C01819=1039.319,-74.831,422.675,168.772,36.713,156.907
C01820=1039.313,-75.080,422.686,168.769,36.713,156.907
C01821=1039.306,-75.330,422.697,168.767,36.713,156.907
C01822=1039.301,-75.580,422.708,168.764,36.713,156.907
C01823=1039.294,-75.829,422.720,168.762,36.713,156.907
C01824=1039.288,-76.079,422.731,168.759,36.713,156.907
C01825=1039.282,-76.329,422.742,168.757,36.713,156.907
C01826=1039.276,-76.578,422.754,168.754,36.713,156.907
C01827=1039.269,-76.828,422.765,168.752,36.714,156.907
C01828=1039.264,-77.077,422.776,168.749,36.714,156.907
C01829=1039.257,-77.328,422.787,168.747,36.714,156.907
C01830=1039.251,-77.576,422.799,168.745,36.714,156.907
C01831=1039.244,-77.826,422.810,168.742,36.714,156.907
C01832=1039.238,-78.076,422.820,168.740,36.714,156.907
C01833=1039.232,-78.326,422.832,168.737,36.714,156.907
C01834=1039.226,-78.575,422.843,168.735,36.714,156.907
C01835=1039.220,-78.825,422.854,168.732,36.714,156.907
C01836=1039.214,-79.075,422.865,168.730,36.714,156.907
C01837=1039.208,-79.325,422.877,168.727,36.714,156.907
C01838=1039.202,-79.574,422.887,168.725,36.714,156.907
C01839=1039.196,-79.824,422.899,168.722,36.714,156.907
C01840=1039.190,-80.074,422.910,168.720,36.714,156.907
C01841=1039.182,-80.323,422.921,168.717,36.714,156.907
C01842=1039.177,-80.573,422.932,168.715,36.714,156.907
C01843=1039.170,-80.823,422.943,168.712,36.714,156.907
C01844=1039.164,-81.072,422.953,168.710,36.714,156.907
C01845=1039.158,-81.321,422.964,168.707,36.715,156.907
C01846=1039.152,-81.572,422.975,168.705,36.715,156.907
C01847=1039.145,-81.821,422.986,168.702,36.715,156.907
C01848=1039.139,-82.071,422.997,168.700,36.715,156.907
C01849=1039.133,-82.321,423.008,168.697,36.716,156.908
C01850=1039.126,-82.570,423.019,168.695,36.716,156.908
C01851=1039.120,-82.820,423.029,168.692,36.716,156.908
C01852=1039.114,-83.070,423.041,168.690,36.716,156.908
C01853=1039.108,-83.319,423.051,168.687,36.716,156.908
C01854=1039.101,-83.605,423.064,168.684,36.716,156.908
C01855=1039.094,-83.889,423.076,168.682,36.717,156.908
C01856=1039.087,-84.174,423.089,168.679,36.717,156.908
C01857=1039.080,-84.459,423.101,168.676,36.717,156.908
C01858=1039.073,-84.709,423.111,168.673,36.717,156.908
C01859=1039.067,-84.958,423.122,168.672,36.718,156.908
C01860=1039.061,-85.209,423.133,168.669,36.718,156.908
C01861=1039.054,-85.458,423.144,168.667,36.718,156.908
C01862=1039.049,-85.707,423.155,168.664,36.718,156.908
C01863=1039.042,-85.957,423.166,168.662,36.719,156.908
C01864=1039.036,-86.207,423.175,168.659,36.719,156.908
C01865=1039.030,-86.457,423.186,168.657,36.719,156.908
C01866=1039.024,-86.707,423.198,168.654,36.719,156.908
C01867=1039.018,-86.956,423.208,168.652,36.719,156.908
C01868=1039.012,-87.206,423.219,168.649,36.719,156.908
C01869=1039.005,-87.456,423.230,168.647,36.719,156.908
C01870=1038.999,-87.705,423.240,168.644,36.720,156.908
C01871=1038.993,-87.954,423.251,168.642,36.720,156.908
C01872=1038.986,-88.205,423.261,168.639,36.720,156.908
C01873=1038.981,-88.454,423.272,168.637,36.721,156.908
C01874=1038.975,-88.704,423.283,168.634,36.721,156.908
C01875=1038.968,-88.954,423.293,168.631,36.721,156.908
C01876=1038.962,-89.203,423.304,168.629,36.721,156.908
C01877=1038.957,-89.453,423.315,168.626,36.721,156.908
C01878=1038.950,-89.703,423.325,168.624,36.721,156.908
C01879=1038.944,-89.953,423.336,168.621,36.722,156.908
C01880=1038.937,-90.202,423.346,168.619,36.722,156.908
C01881=1038.932,-90.451,423.357,168.616,36.722,156.908
C01882=1038.926,-90.702,423.368,168.614,36.723,156.909
C01883=1038.919,-90.951,423.378,168.611,36.723,156.909
C01884=1038.913,-91.201,423.389,168.609,36.723,156.909
C01885=1038.907,-91.450,423.399,168.606,36.723,156.909
C01886=1038.902,-91.700,423.409,168.604,36.723,156.909
C01887=1038.895,-91.950,423.421,168.601,36.724,156.909
C01888=1038.889,-92.200,423.431,168.599,36.724,156.909
C01889=1038.883,-92.450,423.441,168.596,36.724,156.909
C01890=1038.877,-92.699,423.451,168.593,36.725,156.909
C01891=1038.870,-92.949,423.463,168.591,36.725,156.909
C01892=1038.864,-93.199,423.472,168.588,36.725,156.909
C01893=1038.859,-93.448,423.483,168.586,36.726,156.909
C01894=1038.853,-93.698,423.494,168.583,36.726,156.909
C01895=1038.847,-93.948,423.503,168.581,36.726,156.909
C01896=1038.841,-94.197,423.514,168.578,36.726,156.909
C01897=1038.834,-94.447,423.525,168.576,36.726,156.909
C01898=1038.828,-94.697,423.535,168.573,36.727,156.909
C01899=1038.823,-94.947,423.546,168.571,36.727,156.909
C01900=1038.816,-95.196,423.556,168.568,36.727,156.909
C01901=1038.811,-95.446,423.566,168.566,36.728,156.909
C01902=1038.804,-95.695,423.577,168.563,36.728,156.909
C01903=1038.799,-95.945,423.587,168.561,36.728,156.909
C01904=1038.792,-96.195,423.598,168.559,36.728,156.909
C01905=1038.786,-96.445,423.608,168.556,36.728,156.909
C01906=1038.780,-96.694,423.618,168.554,36.729,156.909
C01907=1038.774,-96.944,423.628,168.551,36.729,156.909
C01908=1038.769,-97.194,423.639,168.549,36.730,156.910
C01909=1038.762,-97.443,423.649,168.546,36.730,156.910
C01910=1038.756,-97.693,423.659,168.544,36.730,156.910
C01911=1038.751,-97.943,423.669,168.541,36.730,156.910
C01912=1038.744,-98.193,423.680,168.538,36.731,156.910
C01913=1038.737,-98.443,423.689,168.536,36.731,156.910
C01914=1038.732,-98.692,423.700,168.533,36.732,156.910
C01915=1038.725,-98.942,423.710,168.531,36.732,156.910
C01916=1038.719,-99.191,423.720,168.528,36.732,156.910
C01917=1038.714,-99.441,423.730,168.525,36.733,156.910
C01918=1038.706,-99.729,423.741,168.522,36.734,156.910
C01919=1038.699,-100.015,423.753,168.519,36.734,156.910
C01920=1038.692,-100.303,423.765,168.517,36.734,156.910
C01921=1038.685,-100.590,423.776,168.514,36.735,156.910
C01922=1038.679,-100.840,423.786,168.511,36.735,156.910
C01923=1038.673,-101.089,423.797,168.508,36.736,156.911
C01924=1038.667,-101.339,423.806,168.506,36.737,156.911
C01925=1038.660,-101.589,423.816,168.503,36.737,156.911
C01926=1038.655,-101.839,423.827,168.501,36.737,156.911
C01927=1038.649,-102.088,423.836,168.498,36.737,156.911
C01928=1038.642,-102.338,423.846,168.495,36.738,156.911
C01929=1038.636,-102.587,423.856,168.494,36.739,156.911
C01930=1038.630,-102.837,423.866,168.491,36.739,156.911
C01931=1038.624,-103.087,423.876,168.489,36.739,156.911
C01932=1038.618,-103.336,423.886,168.486,36.740,156.911
C01933=1038.612,-103.587,423.896,168.483,36.740,156.911
C01934=1038.606,-103.836,423.906,168.481,36.741,156.911
C01935=1038.600,-104.086,423.916,168.478,36.741,156.911
C01936=1038.594,-104.335,423.926,168.476,36.741,156.911
C01937=1038.588,-104.585,423.936,168.473,36.742,156.911
C01938=1038.582,-104.835,423.946,168.470,36.743,156.912
C01939=1038.576,-105.085,423.955,168.468,36.743,156.912
C01940=1038.570,-105.335,423.965,168.465,36.743,156.912
C01941=1038.564,-105.584,423.976,168.463,36.744,156.912
C01942=1038.558,-105.834,423.985,168.460,36.745,156.912
C01943=1038.552,-106.084,423.995,168.457,36.745,156.912
C01944=1038.545,-106.334,424.004,168.455,36.745,156.912
C01945=1038.539,-106.583,424.014,168.452,36.746,156.912
C01946=1038.533,-106.833,424.025,168.449,36.747,156.912
C01947=1038.527,-107.083,424.034,168.447,36.747,156.912
C01948=1038.521,-107.333,424.044,168.444,36.747,156.912
C01949=1038.515,-107.582,424.053,168.442,36.748,156.912
C01950=1038.509,-107.832,424.063,168.440,36.749,156.913
C01951=1038.503,-108.082,424.073,168.437,36.749,156.913
C01952=1038.496,-108.332,424.082,168.435,36.749,156.913
C01953=1038.490,-108.582,424.092,168.432,36.750,156.913
C01954=1038.484,-108.831,424.101,168.429,36.751,156.913
C01955=1038.479,-109.081,424.111,168.427,36.751,156.913
C01956=1038.473,-109.331,424.121,168.424,36.752,156.913
C01957=1038.467,-109.580,424.130,168.422,36.753,156.913
C01958=1038.461,-109.830,424.140,168.419,36.753,156.913
C01959=1038.454,-110.079,424.150,168.416,36.754,156.913
C01960=1038.448,-110.329,424.160,168.414,36.754,156.913
C01961=1038.442,-110.579,424.169,168.411,36.755,156.914
C01962=1038.436,-110.829,424.179,168.408,36.756,156.914
C01963=1038.430,-111.079,424.188,168.406,36.756,156.914
C01964=1038.424,-111.329,424.197,168.403,36.757,156.914
C01965=1038.418,-111.579,424.207,168.400,36.757,156.914
C01966=1038.412,-111.828,424.216,168.398,36.758,156.914
C01967=1038.406,-112.078,424.226,168.395,36.758,156.914
C01968=1038.400,-112.327,424.235,168.393,36.759,156.914
C01969=1038.393,-112.577,424.245,168.391,36.760,156.914
C01970=1038.387,-112.827,424.254,168.388,36.760,156.914
C01971=1038.381,-113.077,424.264,168.386,36.761,156.914
C01972=1038.376,-113.326,424.273,168.383,36.762,156.915
C01973=1038.369,-113.576,424.283,168.380,36.762,156.915
C01974=1038.363,-113.826,424.292,168.378,36.762,156.915
C01975=1038.358,-114.076,424.302,168.375,36.763,156.915
C01976=1038.352,-114.325,424.312,168.372,36.764,156.915
C01977=1038.345,-114.576,424.320,168.370,36.764,156.915
C01978=1038.339,-114.825,424.329,168.367,36.765,156.915
C01979=1038.333,-115.074,424.339,168.364,36.766,156.915
C01980=1038.327,-115.324,424.348,168.362,36.766,156.915
C01981=1038.321,-115.574,424.358,168.359,36.767,156.915
C01982=1038.314,-115.861,424.369,168.356,36.768,156.916
C01983=1038.307,-116.147,424.379,168.354,36.769,156.916
C01984=1038.301,-116.433,424.390,168.351,36.770,156.916
C01985=1038.294,-116.719,424.401,168.348,36.770,156.916
C01986=1038.288,-116.969,424.410,168.345,36.771,156.916
C01987=1038.282,-117.219,424.420,168.342,36.772,156.916
C01988=1038.275,-117.469,424.428,168.340,36.772,156.916
C01989=1038.269,-117.718,424.437,168.337,36.773,156.916
C01990=1038.263,-117.968,424.447,168.334,36.774,156.917
C01991=1038.257,-118.218,424.456,168.332,36.774,156.917
C01992=1038.251,-118.468,424.465,168.329,36.775,156.917
C01993=1038.246,-118.717,424.474,168.326,36.776,156.917
C01994=1038.239,-118.967,424.484,168.324,36.777,156.917
C01995=1038.233,-119.217,424.492,168.321,36.777,156.917
C01996=1038.227,-119.467,424.502,168.319,36.779,156.917
C01997=1038.221,-119.716,424.511,168.317,36.779,156.917
C01998=1038.215,-119.967,424.520,168.314,36.780,156.917
C01999=1038.209,-120.216,424.529,168.311,36.781,156.918
C02000=1038.203,-120.465,424.539,168.309,36.781,156.918
C02001=1038.197,-120.716,424.547,168.306,36.782,156.918
C02002=1038.191,-120.965,424.556,168.303,36.783,156.918
C02003=1038.185,-121.216,424.565,168.301,36.783,156.918
C02004=1038.179,-121.465,424.574,168.298,36.784,156.918
C02005=1038.173,-121.715,424.584,168.295,36.785,156.918
C02006=1038.167,-121.965,424.593,168.293,36.786,156.918
C02007=1038.161,-122.214,424.601,168.290,36.787,156.919
C02008=1038.155,-122.464,424.610,168.287,36.787,156.919
C02009=1038.149,-122.714,424.620,168.286,36.788,156.919
C02010=1038.143,-122.963,424.629,168.283,36.789,156.919
C02011=1038.137,-123.213,424.637,168.280,36.789,156.919
C02012=1038.131,-123.463,424.647,168.277,36.791,156.919
C02013=1038.125,-123.713,424.655,168.275,36.791,156.919
C02014=1038.119,-123.963,424.665,168.272,36.792,156.919
C02015=1038.114,-124.212,424.673,168.269,36.793,156.920
C02016=1038.107,-124.462,424.682,168.267,36.793,156.920
C02017=1038.101,-124.712,424.691,168.264,36.794,156.920
C02018=1038.095,-124.961,424.700,168.261,36.795,156.920
C02019=1038.089,-125.211,424.709,168.259,36.796,156.920
C02020=1038.083,-125.461,424.718,168.256,36.797,156.920
C02021=1038.077,-125.711,424.727,168.254,36.798,156.920
C02022=1038.071,-125.961,424.735,168.251,36.799,156.920
C02023=1038.065,-126.210,424.744,168.249,36.800,156.921
C02024=1038.059,-126.461,424.753,168.246,36.800,156.921
C02025=1038.053,-126.710,424.762,168.243,36.802,156.921
C02026=1038.047,-126.960,424.770,168.241,36.802,156.921
C02027=1038.041,-127.210,424.779,168.238,36.803,156.921
C02028=1038.035,-127.459,424.788,168.235,36.804,156.921
C02029=1038.029,-127.709,424.797,168.233,36.805,156.921
C02030=1038.024,-127.958,424.806,168.230,36.806,156.922
C02031=1038.019,-128.208,424.816,168.227,36.806,156.922
C02032=1038.014,-128.458,424.825,168.225,36.806,156.922
C02033=1038.011,-128.708,424.836,168.223,36.805,156.921
C02034=1038.008,-128.958,424.847,168.221,36.804,156.921
C02035=1038.007,-129.208,424.860,168.219,36.802,156.921
C02036=1038.005,-129.458,424.872,168.217,36.800,156.921
C02037=1038.005,-129.707,424.885,168.215,36.798,156.920
C02038=1038.005,-129.957,424.899,168.213,36.794,156.920
C02039=1038.006,-130.208,424.914,168.212,36.791,156.919
C02040=1038.009,-130.458,424.929,168.210,36.787,156.918
C02041=1038.012,-130.707,424.943,168.209,36.783,156.918
C02042=1038.015,-130.959,424.959,168.207,36.779,156.917
C02043=1038.019,-131.208,424.976,168.207,36.773,156.916
C02044=1038.024,-131.459,424.994,168.205,36.767,156.915
C02045=1038.030,-131.708,425.011,168.205,36.761,156.914
C02046=1037.689,-131.732,424.743,168.156,36.967,156.948
C02047=1037.683,-131.483,424.725,168.158,36.973,156.949
C02048=1037.679,-131.233,424.707,168.158,36.978,156.950
C02049=1037.674,-130.983,424.691,168.160,36.984,156.951
C02050=1037.671,-130.732,424.674,168.161,36.988,156.952
C02051=1037.668,-130.483,424.660,168.162,36.993,156.953
C02052=1037.666,-130.232,424.644,168.164,36.997,156.954
C02053=1037.665,-129.982,424.630,168.166,37.000,156.954
C02054=1037.664,-129.732,424.616,168.167,37.003,156.955
C02055=1037.665,-129.482,424.603,168.169,37.006,156.955
C02056=1037.665,-129.232,424.590,168.171,37.007,156.955
C02057=1037.668,-128.983,424.579,168.173,37.009,156.956
C02058=1037.670,-128.733,424.567,168.175,37.010,156.956
C02059=1037.674,-128.483,424.556,168.178,37.011,156.956
C02060=1037.677,-128.232,424.546,168.180,37.011,156.956
C02061=1037.682,-127.983,424.536,168.182,37.011,156.956
C02062=1037.688,-127.734,424.527,168.185,37.010,156.956
C02063=1037.694,-127.484,424.519,168.188,37.009,156.956
C02064=1037.700,-127.234,424.510,168.190,37.009,156.956
C02065=1037.706,-126.984,424.501,168.193,37.007,156.955
C02066=1037.712,-126.735,424.493,168.196,37.007,156.955
C02067=1037.718,-126.485,424.484,168.199,37.006,156.955
C02068=1037.724,-126.234,424.475,168.200,37.004,156.955
C02069=1037.730,-125.986,424.466,168.203,37.004,156.955
C02070=1037.736,-125.735,424.457,168.206,37.003,156.955
C02071=1037.741,-125.486,424.449,168.209,37.002,156.955
C02072=1037.748,-125.236,424.440,168.211,37.001,156.954
C02073=1037.754,-124.986,424.431,168.214,37.000,156.954
C02074=1037.760,-124.737,424.422,168.217,37.000,156.954
C02075=1037.766,-124.486,424.413,168.219,36.998,156.954
C02076=1037.772,-124.237,424.404,168.222,36.998,156.954
C02077=1037.778,-123.987,424.395,168.225,36.997,156.954
C02078=1037.784,-123.737,424.386,168.228,36.996,156.954
C02079=1037.790,-123.488,424.378,168.229,36.995,156.953
C02080=1037.796,-123.238,424.368,168.232,36.994,156.953
C02081=1037.802,-122.987,424.360,168.235,36.993,156.953
C02082=1037.808,-122.738,424.350,168.237,36.993,156.953
C02083=1037.814,-122.488,424.342,168.240,36.992,156.953
C02084=1037.820,-122.238,424.332,168.243,36.991,156.953
C02085=1037.826,-121.989,424.324,168.245,36.990,156.953
C02086=1037.832,-121.739,424.314,168.248,36.989,156.953
C02087=1037.838,-121.489,424.305,168.251,36.989,156.953
C02088=1037.844,-121.240,424.297,168.254,36.988,156.952
C02089=1037.850,-120.990,424.287,168.256,36.987,156.952
C02090=1037.856,-120.740,424.279,168.258,36.986,156.952
C02091=1037.861,-120.490,424.269,168.261,36.985,156.952
C02092=1037.868,-120.241,424.260,168.263,36.984,156.952
C02093=1037.874,-119.990,424.251,168.266,36.984,156.952
C02094=1037.880,-119.741,424.242,168.269,36.983,156.952
C02095=1037.886,-119.492,424.233,168.271,36.982,156.952
C02096=1037.892,-119.241,424.224,168.274,36.982,156.952
C02097=1037.898,-118.991,424.214,168.277,36.980,156.951
C02098=1037.904,-118.742,424.205,168.280,36.980,156.951
C02099=1037.909,-118.492,424.196,168.282,36.979,156.951
C02100=1037.916,-118.242,424.187,168.285,36.978,156.951
C02101=1037.923,-117.993,424.178,168.288,36.978,156.951
C02102=1037.928,-117.744,424.169,168.290,36.977,156.951
C02103=1037.934,-117.493,424.160,168.292,36.976,156.951
C02104=1037.940,-117.243,424.150,168.295,36.975,156.951
C02105=1037.946,-116.994,424.141,168.297,36.975,156.950
C02106=1037.952,-116.744,424.132,168.300,36.974,156.950
C02107=1037.959,-116.458,424.121,168.303,36.973,156.950
C02108=1037.966,-116.172,424.110,168.306,36.972,156.950
C02109=1037.973,-115.885,424.099,168.309,36.971,156.950
C02110=1037.980,-115.599,424.089,168.312,36.971,156.950
C02111=1037.986,-115.349,424.080,168.315,36.970,156.950
C02112=1037.992,-115.099,424.071,168.318,36.969,156.950
C02113=1037.998,-114.849,424.061,168.320,36.969,156.950
C02114=1038.004,-114.600,424.052,168.323,36.968,156.949
C02115=1038.010,-114.350,424.042,168.326,36.967,156.949
C02116=1038.016,-114.100,424.033,168.327,36.967,156.949
C02117=1038.022,-113.851,424.024,168.330,36.966,156.949
C02118=1038.028,-113.600,424.015,168.333,36.965,156.949
C02119=1038.034,-113.351,424.005,168.335,36.964,156.949
C02120=1038.040,-113.101,423.996,168.338,36.964,156.949
C02121=1038.046,-112.851,423.986,168.341,36.963,156.949
C02122=1038.052,-112.601,423.976,168.343,36.962,156.949
C02123=1038.058,-112.352,423.967,168.346,36.962,156.948
C02124=1038.064,-112.102,423.958,168.349,36.961,156.948
C02125=1038.070,-111.853,423.948,168.351,36.960,156.948
C02126=1038.077,-111.603,423.939,168.354,36.960,156.948
C02127=1038.083,-111.353,423.929,168.357,36.959,156.948
C02128=1038.089,-111.103,423.919,168.359,36.958,156.948
C02129=1038.095,-110.853,423.910,168.362,36.958,156.948
C02130=1038.101,-110.604,423.900,168.365,36.957,156.948
C02131=1038.106,-110.354,423.890,168.366,36.957,156.948
C02132=1038.112,-110.104,423.881,168.369,36.956,156.948
C02133=1038.118,-109.855,423.871,168.372,36.955,156.948
C02134=1038.125,-109.605,423.862,168.374,36.955,156.947
C02135=1038.131,-109.355,423.852,168.377,36.954,156.947
C02136=1038.137,-109.105,423.843,168.380,36.953,156.947
C02137=1038.143,-108.855,423.833,168.382,36.953,156.947
C02138=1038.149,-108.606,423.824,168.385,36.952,156.947
C02139=1038.155,-108.356,423.814,168.388,36.952,156.947
C02140=1038.162,-108.106,423.804,168.390,36.951,156.947
C02141=1038.168,-107.856,423.795,168.393,36.951,156.947
C02142=1038.174,-107.606,423.785,168.396,36.950,156.947
C02143=1038.180,-107.357,423.776,168.398,36.949,156.947
C02144=1038.185,-107.107,423.766,168.401,36.949,156.947
C02145=1038.191,-106.858,423.756,168.403,36.948,156.947
C02146=1038.198,-106.608,423.746,168.406,36.948,156.946
C02147=1038.204,-106.358,423.736,168.409,36.947,156.946
C02148=1038.210,-106.109,423.727,168.410,36.946,156.946
C02149=1038.215,-105.858,423.717,168.413,36.946,156.946
C02150=1038.222,-105.609,423.707,168.416,36.946,156.946
C02151=1038.228,-105.360,423.697,168.418,36.945,156.946
C02152=1038.234,-105.110,423.687,168.421,36.944,156.946
C02153=1038.240,-104.860,423.677,168.423,36.944,156.946
C02154=1038.246,-104.610,423.668,168.426,36.944,156.946
C02155=1038.252,-104.360,423.658,168.429,36.943,156.946
C02156=1038.258,-104.111,423.648,168.431,36.942,156.946
C02157=1038.264,-103.861,423.638,168.434,36.942,156.946
C02158=1038.270,-103.611,423.628,168.437,36.942,156.945
C02159=1038.276,-103.361,423.618,168.439,36.941,156.945
C02160=1038.283,-103.112,423.608,168.442,36.940,156.945
C02161=1038.288,-102.862,423.598,168.444,36.940,156.945
C02162=1038.294,-102.612,423.588,168.447,36.939,156.945
C02163=1038.301,-102.363,423.578,168.450,36.939,156.945
C02164=1038.307,-102.113,423.569,168.452,36.939,156.945
C02165=1038.312,-101.863,423.558,168.455,36.938,156.945
C02166=1038.319,-101.614,423.548,168.457,36.937,156.945
C02167=1038.325,-101.364,423.539,168.460,36.937,156.945
C02168=1038.331,-101.114,423.528,168.462,36.937,156.945
C02169=1038.338,-100.864,423.518,168.464,36.936,156.945
C02170=1038.344,-100.614,423.508,168.467,36.936,156.945
C02171=1038.350,-100.327,423.497,168.470,36.935,156.945
C02172=1038.357,-100.040,423.485,168.473,36.935,156.944
C02173=1038.365,-99.753,423.474,168.476,36.934,156.944
C02174=1038.371,-99.466,423.462,168.479,36.933,156.944
C02175=1038.377,-99.216,423.452,168.482,36.933,156.944
C02176=1038.384,-98.967,423.442,168.484,36.932,156.944
C02177=1038.389,-98.717,423.432,168.487,36.932,156.944
C02178=1038.396,-98.466,423.422,168.489,36.932,156.944
C02179=1038.403,-98.217,423.411,168.492,36.931,156.944
C02180=1038.409,-97.967,423.402,168.495,36.931,156.944
C02181=1038.414,-97.718,423.391,168.497,36.930,156.944
C02182=1038.421,-97.468,423.381,168.500,36.930,156.944
C02183=1038.426,-97.218,423.371,168.502,36.930,156.944
C02184=1038.433,-96.968,423.361,168.505,36.929,156.944
C02185=1038.438,-96.719,423.350,168.507,36.929,156.944
C02186=1038.444,-96.469,423.341,168.510,36.928,156.944
C02187=1038.451,-96.219,423.329,168.513,36.928,156.944
C02188=1038.457,-95.970,423.319,168.515,36.928,156.944
C02189=1038.463,-95.720,423.309,168.518,36.927,156.943
C02190=1038.468,-95.470,423.298,168.520,36.927,156.943
C02191=1038.475,-95.220,423.288,168.523,36.927,156.943
C02192=1038.480,-94.971,423.278,168.525,36.927,156.943
C02193=1038.487,-94.721,423.268,168.527,36.926,156.943
C02194=1038.493,-94.471,423.257,168.530,36.926,156.943
C02195=1038.499,-94.222,423.246,168.532,36.925,156.943
C02196=1038.505,-93.972,423.236,168.535,36.925,156.943
C02197=1038.511,-93.722,423.225,168.537,36.925,156.943
C02198=1038.517,-93.473,423.215,168.540,36.925,156.943
C02199=1038.522,-93.223,423.205,168.542,36.925,156.943
C02200=1038.530,-92.973,423.194,168.545,36.924,156.943
C02201=1038.535,-92.724,423.183,168.547,36.924,156.943
C02202=1038.541,-92.473,423.173,168.550,36.923,156.943
C02203=1038.547,-92.224,423.163,168.553,36.923,156.943
C02204=1038.553,-91.975,423.152,168.555,36.923,156.943
C02205=1038.560,-91.724,423.142,168.558,36.922,156.943
C02206=1038.565,-91.475,423.131,168.560,36.922,156.943
C02207=1038.572,-91.226,423.121,168.563,36.922,156.943
C02208=1038.578,-90.976,423.110,168.565,36.922,156.943
C02209=1038.584,-90.725,423.100,168.568,36.922,156.943
C02210=1038.590,-90.476,423.089,168.570,36.921,156.943
C02211=1038.596,-90.227,423.078,168.573,36.921,156.943
C02212=1038.602,-89.977,423.068,168.576,36.920,156.943
C02213=1038.608,-89.727,423.058,168.578,36.920,156.943
C02214=1038.614,-89.477,423.047,168.581,36.920,156.943
C02215=1038.621,-89.228,423.037,168.583,36.920,156.942
C02216=1038.626,-88.978,423.026,168.586,36.919,156.942
C02217=1038.632,-88.728,423.015,168.588,36.919,156.942
C02218=1038.639,-88.478,423.005,168.591,36.919,156.942
C02219=1038.645,-88.229,422.994,168.593,36.919,156.942
C02220=1038.652,-87.979,422.983,168.596,36.918,156.942
C02221=1038.657,-87.730,422.972,168.598,36.918,156.942
C02222=1038.663,-87.480,422.962,168.601,36.918,156.942
C02223=1038.670,-87.230,422.952,168.603,36.917,156.942
C02224=1038.676,-86.980,422.941,168.606,36.917,156.942
C02225=1038.681,-86.731,422.930,168.609,36.917,156.942
C02226=1038.688,-86.481,422.919,168.611,36.917,156.942
C02227=1038.694,-86.231,422.908,168.614,36.917,156.942
C02228=1038.700,-85.982,422.897,168.616,36.917,156.942
C02229=1038.707,-85.732,422.887,168.619,36.916,156.942
C02230=1038.713,-85.482,422.876,168.621,36.916,156.942
C02231=1038.719,-85.233,422.866,168.624,36.916,156.942
C02232=1038.726,-84.983,422.854,168.625,36.915,156.942
C02233=1038.731,-84.734,422.844,168.628,36.915,156.942
C02234=1038.738,-84.484,422.834,168.630,36.915,156.942
C02235=1038.745,-84.199,422.821,168.633,36.914,156.942
C02236=1038.752,-83.913,422.808,168.636,36.914,156.942
C02237=1038.758,-83.629,422.796,168.639,36.914,156.942
C02238=1038.766,-83.343,422.784,168.642,36.914,156.942
C02239=1038.772,-83.094,422.774,168.644,36.914,156.942
C02240=1038.779,-82.844,422.762,168.647,36.913,156.942
C02241=1038.784,-82.594,422.751,168.650,36.913,156.942
C02242=1038.791,-82.345,422.741,168.652,36.913,156.942
C02243=1038.797,-82.095,422.730,168.655,36.913,156.942
C02244=1038.804,-81.845,422.719,168.657,36.912,156.941
C02245=1038.810,-81.596,422.708,168.660,36.912,156.941
C02246=1038.816,-81.346,422.697,168.662,36.912,156.941
C02247=1038.822,-81.096,422.686,168.665,36.911,156.941
C02248=1038.829,-80.848,422.675,168.667,36.911,156.941
C02249=1038.835,-80.597,422.664,168.670,36.911,156.941
C02250=1038.841,-80.348,422.653,168.672,36.911,156.941
C02251=1038.847,-80.098,422.642,168.675,36.911,156.941
C02252=1038.854,-79.848,422.632,168.677,36.911,156.941
C02253=1038.860,-79.598,422.620,168.680,36.911,156.941
C02254=1038.866,-79.349,422.609,168.682,36.911,156.941
C02255=1038.872,-79.099,422.598,168.685,36.911,156.941
C02256=1038.878,-78.850,422.587,168.687,36.910,156.941
C02257=1038.885,-78.600,422.575,168.690,36.910,156.941
C02258=1038.890,-78.350,422.565,168.692,36.910,156.941
C02259=1038.897,-78.100,422.553,168.695,36.910,156.941
C02260=1038.902,-77.850,422.542,168.697,36.910,156.941
C02261=1038.909,-77.601,422.530,168.700,36.910,156.941
C02262=1038.915,-77.352,422.520,168.702,36.910,156.941
C02263=1038.922,-77.101,422.509,168.705,36.910,156.941
C02264=1038.928,-76.852,422.498,168.707,36.910,156.941
C02265=1038.934,-76.602,422.486,168.709,36.909,156.941
C02266=1038.940,-76.353,422.475,168.712,36.909,156.941
C02267=1038.946,-76.103,422.464,168.714,36.909,156.941
C02268=1038.952,-75.853,422.453,168.717,36.909,156.941
C02269=1038.959,-75.604,422.441,168.719,36.909,156.941
C02270=1038.964,-75.354,422.430,168.722,36.909,156.941
C02271=1038.971,-75.104,422.419,168.724,36.909,156.941
C02272=1038.977,-74.855,422.407,168.727,36.909,156.941
C02273=1038.983,-74.605,422.396,168.729,36.909,156.941
C02274=1038.989,-74.355,422.385,168.732,36.909,156.941
C02275=1038.996,-74.106,422.373,168.734,36.909,156.941
C02276=1039.002,-73.856,422.362,168.737,36.909,156.941
C02277=1039.008,-73.606,422.351,168.739,36.909,156.941
C02278=1039.014,-73.357,422.339,168.741,36.909,156.941
C02279=1039.019,-73.107,422.328,168.744,36.909,156.941
C02280=1039.026,-72.857,422.316,168.746,36.909,156.941
C02281=1039.032,-72.608,422.305,168.749,36.909,156.941
C02282=1039.038,-72.358,422.293,168.751,36.909,156.941
C02283=1039.044,-72.109,422.282,168.754,36.909,156.941
C02284=1039.050,-71.859,422.270,168.756,36.909,156.941
C02285=1039.056,-71.609,422.259,168.758,36.909,156.941
C02286=1039.062,-71.359,422.247,168.761,36.909,156.941
C02287=1039.069,-71.109,422.235,168.763,36.909,156.941
C02288=1039.074,-70.860,422.224,168.766,36.909,156.941
C02289=1039.080,-70.610,422.212,168.768,36.909,156.941
C02290=1039.086,-70.361,422.200,168.770,36.909,156.941
C02291=1039.093,-70.111,422.189,168.773,36.909,156.941
C02292=1039.099,-69.861,422.177,168.775,36.910,156.942
C02293=1039.104,-69.612,422.166,168.778,36.910,156.942
C02294=1039.111,-69.362,422.154,168.780,36.910,156.942
C02295=1039.117,-69.113,422.143,168.782,36.910,156.942
C02296=1039.123,-68.863,422.131,168.785,36.910,156.942
C02297=1039.129,-68.613,422.119,168.787,36.909,156.942
C02298=1039.135,-68.364,422.108,168.790,36.909,156.942
C02299=1039.142,-68.080,422.094,168.792,36.910,156.942
C02300=1039.149,-67.798,422.081,168.795,36.910,156.942
C02301=1039.156,-67.515,422.068,168.798,36.910,156.942
C02302=1039.163,-67.233,422.054,168.801,36.910,156.942
C02303=1039.169,-66.983,422.043,168.803,36.910,156.942
C02304=1039.175,-66.733,422.031,168.805,36.910,156.942
C02305=1039.181,-66.484,422.019,168.808,36.911,156.942
C02306=1039.188,-66.234,422.008,168.810,36.911,156.942
C02307=1039.194,-65.984,421.996,168.813,36.911,156.942
C02308=1039.200,-65.734,421.983,168.815,36.910,156.942
C02309=1039.206,-65.485,421.972,168.817,36.910,156.942
C02310=1039.212,-65.235,421.960,168.820,36.910,156.942
C02311=1039.219,-64.986,421.949,168.823,36.911,156.942
C02312=1039.224,-64.736,421.937,168.826,36.911,156.942
C02313=1039.231,-64.486,421.925,168.828,36.911,156.942
C02314=1039.237,-64.237,421.913,168.830,36.911,156.942
C02315=1039.243,-63.987,421.901,168.833,36.911,156.942
C02316=1039.249,-63.737,421.890,168.835,36.911,156.942
C02317=1039.256,-63.488,421.878,168.837,36.912,156.942
C02318=1039.262,-63.238,421.866,168.840,36.912,156.942
C02319=1039.268,-62.988,421.853,168.842,36.912,156.942
C02320=1039.274,-62.739,421.842,168.845,36.911,156.942
C02321=1039.281,-62.489,421.830,168.847,36.911,156.942
C02322=1039.287,-62.239,421.818,168.849,36.912,156.942
C02323=1039.293,-61.990,421.806,168.852,36.912,156.942
C02324=1039.299,-61.741,421.794,168.854,36.912,156.942
C02325=1039.305,-61.490,421.782,168.857,36.912,156.942
C02326=1039.312,-61.241,421.770,168.859,36.912,156.942
C02327=1039.318,-60.991,421.759,168.861,36.913,156.942
C02328=1039.325,-60.742,421.747,168.864,36.913,156.942
C02329=1039.330,-60.493,421.734,168.866,36.913,156.942
C02330=1039.337,-60.243,421.722,168.868,36.913,156.942
C02331=1039.343,-59.993,421.711,168.871,36.913,156.942
C02332=1039.349,-59.743,421.699,168.873,36.913,156.943
C02333=1039.356,-59.493,421.687,168.876,36.913,156.943
C02334=1039.362,-59.244,421.675,168.878,36.913,156.943
C02335=1039.368,-58.995,421.663,168.880,36.913,156.943
C02336=1039.374,-58.745,421.651,168.883,36.914,156.943
C02337=1039.381,-58.495,421.639,168.885,36.914,156.943
C02338=1039.387,-58.246,421.626,168.887,36.914,156.943
C02339=1039.393,-57.996,421.614,168.890,36.914,156.943
C02340=1039.400,-57.746,421.602,168.892,36.914,156.943
C02341=1039.406,-57.496,421.590,168.895,36.914,156.943
C02342=1039.412,-57.246,421.578,168.897,36.914,156.943
C02343=1039.418,-56.997,421.567,168.899,36.914,156.943
C02344=1039.424,-56.748,421.554,168.902,36.914,156.943
C02345=1039.431,-56.498,421.542,168.904,36.915,156.943
C02346=1039.438,-56.248,421.530,168.906,36.915,156.943
C02347=1039.444,-55.999,421.518,168.909,36.915,156.943
C02348=1039.450,-55.749,421.506,168.911,36.915,156.943
C02349=1039.457,-55.499,421.494,168.913,36.915,156.943
C02350=1039.463,-55.249,421.481,168.916,36.915,156.943
C02351=1039.469,-55.000,421.469,168.918,36.915,156.943
C02352=1039.476,-54.751,421.456,168.921,36.915,156.943
C02353=1039.482,-54.501,421.444,168.923,36.915,156.943
C02354=1039.489,-54.252,421.432,168.925,36.916,156.943
C02355=1039.495,-54.002,421.420,168.928,36.916,156.943
C02356=1039.501,-53.753,421.408,168.930,36.916,156.943
C02357=1039.507,-53.503,421.396,168.932,36.916,156.943
C02358=1039.513,-53.253,421.383,168.935,36.916,156.943
C02359=1039.520,-53.004,421.371,168.937,36.916,156.943
C02360=1039.527,-52.754,421.360,168.939,36.916,156.943
C02361=1039.533,-52.504,421.347,168.943,36.916,156.943
C02362=1039.539,-52.255,421.335,168.945,36.917,156.944
C02363=1039.547,-51.973,421.321,168.948,36.917,156.944
C02364=1039.554,-51.691,421.307,168.950,36.917,156.944
C02365=1039.561,-51.410,421.292,168.953,36.917,156.944
C02366=1039.569,-51.128,421.279,168.956,36.917,156.944
C02367=1039.575,-50.879,421.266,168.958,36.917,156.944
C02368=1039.582,-50.629,421.254,168.960,36.917,156.944
C02369=1039.588,-50.379,421.242,168.963,36.918,156.944
C02370=1039.593,-50.129,421.229,168.965,36.918,156.944
C02371=1039.600,-49.880,421.217,168.967,36.919,156.944
C02372=1039.606,-49.631,421.204,168.969,36.919,156.944
C02373=1039.612,-49.381,421.191,168.972,36.919,156.944
C02374=1039.619,-49.131,421.179,168.974,36.919,156.944
C02375=1039.625,-48.882,421.166,168.976,36.920,156.944
C02376=1039.631,-48.632,421.153,168.979,36.920,156.944
C02377=1039.637,-48.382,421.141,168.981,36.920,156.944
C02378=1039.644,-48.133,421.129,168.983,36.920,156.944
C02379=1039.650,-47.883,421.116,168.985,36.921,156.945
C02380=1039.656,-47.633,421.103,168.988,36.921,156.945
C02381=1039.662,-47.384,421.090,168.990,36.922,156.945
C02382=1039.669,-47.135,421.078,168.992,36.922,156.945
C02383=1039.674,-46.885,421.065,168.995,36.922,156.945
C02384=1039.681,-46.635,421.052,168.997,36.922,156.945
C02385=1039.687,-46.386,421.039,168.999,36.923,156.945
C02386=1039.693,-46.136,421.028,169.001,36.923,156.945
C02387=1039.699,-45.887,421.014,169.005,36.923,156.945
C02388=1039.705,-45.637,421.002,169.007,36.924,156.945
C02389=1039.712,-45.388,420.988,169.009,36.924,156.945
C02390=1039.718,-45.138,420.976,169.011,36.925,156.945
C02391=1039.724,-44.888,420.964,169.014,36.925,156.945
C02392=1039.730,-44.639,420.951,169.016,36.925,156.945
C02393=1039.736,-44.389,420.938,169.018,36.925,156.945
C02394=1039.743,-44.140,420.925,169.020,36.926,156.946
C02395=1039.749,-43.890,420.913,169.023,36.926,156.946
C02396=1039.756,-43.640,420.899,169.025,36.926,156.946
C02397=1039.762,-43.390,420.887,169.027,36.926,156.946
C02398=1039.769,-43.141,420.874,169.030,36.927,156.946
C02399=1039.775,-42.891,420.861,169.032,36.927,156.946
C02400=1039.781,-42.642,420.848,169.034,36.928,156.946
C02401=1039.787,-42.392,420.836,169.036,36.928,156.946
C02402=1039.793,-42.143,420.822,169.039,36.928,156.946
C02403=1039.800,-41.894,420.810,169.041,36.928,156.946
C02404=1039.806,-41.644,420.797,169.043,36.929,156.946
C02405=1039.812,-41.394,420.784,169.045,36.929,156.946
C02406=1039.819,-41.144,420.771,169.048,36.929,156.946
C02407=1039.825,-40.895,420.759,169.050,36.930,156.946
C02408=1039.831,-40.646,420.746,169.052,36.930,156.946
C02409=1039.838,-40.396,420.732,169.055,36.931,156.947
C02410=1039.844,-40.146,420.720,169.058,36.931,156.947
C02411=1039.850,-39.896,420.706,169.060,36.931,156.947
C02412=1039.857,-39.647,420.694,169.062,36.931,156.947
C02413=1039.863,-39.398,420.681,169.064,36.932,156.947
C02414=1039.869,-39.148,420.668,169.067,36.932,156.947
C02415=1039.876,-38.898,420.655,169.069,36.932,156.947
C02416=1039.882,-38.648,420.642,169.071,36.933,156.947
C02417=1039.888,-38.399,420.628,169.073,36.933,156.947
C02418=1039.894,-38.149,420.616,169.075,36.934,156.947
C02419=1039.901,-37.900,420.602,169.078,36.934,156.947
C02420=1039.907,-37.650,420.589,169.080,36.934,156.947
C02421=1039.913,-37.400,420.576,169.082,36.935,156.947
C02422=1039.919,-37.151,420.563,169.084,36.935,156.948
C02423=1039.926,-36.902,420.550,169.086,36.936,156.948
C02424=1039.932,-36.652,420.536,169.089,36.936,156.948
C02425=1039.938,-36.402,420.524,169.091,36.937,156.948
C02426=1039.945,-36.153,420.510,169.093,36.937,156.948
C02427=1039.951,-35.872,420.495,169.096,36.938,156.948
C02428=1039.958,-35.591,420.480,169.098,36.938,156.948
C02429=1039.966,-35.309,420.466,169.101,36.939,156.948
C02430=1039.973,-35.028,420.450,169.104,36.939,156.948
C02431=1039.979,-34.779,420.437,169.106,36.940,156.948
C02432=1039.985,-34.530,420.424,169.108,36.940,156.948
C02433=1039.991,-34.280,420.411,169.111,36.940,156.949
C02434=1039.998,-34.030,420.398,169.113,36.941,156.949
C02435=1040.004,-33.781,420.384,169.115,36.941,156.949
C02436=1040.010,-33.531,420.371,169.117,36.942,156.949
C02437=1040.016,-33.282,420.358,169.119,36.942,156.949
C02438=1040.023,-33.032,420.344,169.121,36.943,156.949
C02439=1040.029,-32.783,420.331,169.124,36.943,156.949
C02440=1040.035,-32.533,420.318,169.126,36.943,156.949
C02441=1040.041,-32.283,420.304,169.128,36.944,156.949
C02442=1040.048,-32.033,420.291,169.130,36.945,156.949
C02443=1040.054,-31.784,420.278,169.132,36.945,156.949
C02444=1040.061,-31.534,420.264,169.135,36.945,156.950
C02445=1040.067,-31.285,420.251,169.138,36.946,156.950
C02446=1040.073,-31.036,420.237,169.140,36.946,156.950
C02447=1040.079,-30.786,420.224,169.142,36.946,156.950
C02448=1040.086,-30.536,420.210,169.144,36.947,156.950
C02449=1040.092,-30.287,420.197,169.146,36.948,156.950
C02450=1040.099,-30.038,420.184,169.149,36.948,156.950
C02451=1040.105,-29.788,420.170,169.151,36.948,156.950
C02452=1040.112,-29.539,420.157,169.153,36.949,156.950
C02453=1040.118,-29.288,420.143,169.155,36.950,156.950
C02454=1040.124,-29.039,420.130,169.157,36.949,156.950
C02455=1040.130,-28.790,420.116,169.159,36.950,156.951
C02456=1040.137,-28.540,420.103,169.162,36.951,156.951
C02457=1040.143,-28.291,420.089,169.164,36.951,156.951
C02458=1040.149,-28.041,420.076,169.166,36.951,156.951
C02459=1040.156,-27.791,420.062,169.168,36.952,156.951
C02460=1040.162,-27.542,420.049,169.170,36.953,156.951
C02461=1040.169,-27.292,420.036,169.172,36.953,156.951
C02462=1040.175,-27.043,420.022,169.176,36.953,156.951
C02463=1040.181,-26.793,420.008,169.178,36.954,156.951
C02464=1040.188,-26.543,419.995,169.180,36.954,156.951
C02465=1040.193,-26.294,419.981,169.182,36.955,156.952
C02466=1040.200,-26.044,419.967,169.184,36.956,156.952
C02467=1040.206,-25.795,419.954,169.186,36.956,156.952
C02468=1040.212,-25.545,419.940,169.188,36.956,156.952
C02469=1040.219,-25.296,419.926,169.191,36.957,156.952
C02470=1040.225,-25.046,419.913,169.193,36.957,156.952
C02471=1040.231,-24.796,419.898,169.195,36.958,156.952
C02472=1040.237,-24.547,419.885,169.197,36.959,156.952
C02473=1040.243,-24.298,419.872,169.199,36.959,156.952
C02474=1040.250,-24.047,419.857,169.201,36.960,156.953
C02475=1040.256,-23.799,419.844,169.204,36.961,156.953
C02476=1040.263,-23.549,419.830,169.206,36.961,156.953
C02477=1040.268,-23.299,419.816,169.208,36.961,156.953
C02478=1040.275,-23.049,419.802,169.211,36.962,156.953
C02479=1040.281,-22.800,419.788,169.213,36.962,156.953
C02480=1040.287,-22.551,419.775,169.215,36.963,156.953
C02481=1040.294,-22.301,419.761,169.217,36.964,156.953
C02482=1040.299,-22.051,419.747,169.219,36.964,156.953
C02483=1040.307,-21.802,419.733,169.221,36.965,156.953
C02484=1040.313,-21.553,419.719,169.223,36.965,156.954
C02485=1040.319,-21.303,419.705,169.225,36.966,156.954
C02486=1040.325,-21.053,419.692,169.227,36.967,156.954
C02487=1040.331,-20.823,419.679,169.229,36.967,156.954
C02488=1040.337,-20.594,419.666,169.231,36.967,156.954
C02489=1040.342,-20.364,419.653,169.233,36.968,156.954
C02490=1040.348,-20.134,419.640,169.236,36.969,156.954
C02491=1040.354,-19.904,419.627,169.238,36.969,156.954
C02492=1040.361,-19.674,419.615,169.240,36.969,156.954
C02493=1040.367,-19.445,419.602,169.242,36.970,156.954
C02494=1040.375,-19.071,419.581,169.245,36.971,156.955
C02495=1040.386,-18.679,419.559,169.248,36.972,156.955
C02496=1040.392,-18.429,419.545,169.251,36.972,156.955
C02497=1040.398,-18.179,419.531,169.253,36.973,156.955
C02498=1040.404,-17.930,419.516,169.255,36.973,156.955
C02499=1040.411,-17.680,419.503,169.257,36.974,156.955
C02500=1040.418,-17.431,419.489,169.259,36.975,156.955
C02501=1040.424,-17.181,419.475,169.261,36.975,156.955
C02502=1040.430,-16.932,419.461,169.263,36.975,156.956
C02503=1040.436,-16.682,419.446,169.266,36.976,156.956
C02504=1040.443,-16.433,419.433,169.268,36.977,156.956
C02505=1040.450,-16.183,419.419,169.270,36.977,156.956
C02506=1040.455,-15.934,419.405,169.273,36.978,156.956
C02507=1040.462,-15.684,419.391,169.275,36.978,156.956
C02508=1040.468,-15.434,419.376,169.277,36.979,156.956
C02509=1040.475,-15.185,419.362,169.279,36.980,156.956
C02510=1040.481,-14.935,419.348,169.281,36.980,156.957
C02511=1040.487,-14.686,419.333,169.283,36.981,156.957
C02512=1040.494,-14.436,419.320,169.285,36.981,156.957
C02513=1040.499,-14.187,419.305,169.287,36.982,156.957
C02514=1040.506,-13.937,419.292,169.289,36.983,156.957
C02515=1040.513,-13.688,419.277,169.292,36.983,156.957
C02516=1040.518,-13.438,419.263,169.294,36.984,156.957
C02517=1040.525,-13.189,419.248,169.296,36.985,156.957
C02518=1040.531,-12.940,419.234,169.298,36.985,156.958
C02519=1040.537,-12.690,419.220,169.300,36.986,156.958
C02520=1040.544,-12.440,419.205,169.302,36.986,156.958
C02521=1040.550,-12.191,419.191,169.304,36.987,156.958
C02522=1040.556,-11.941,419.177,169.306,36.988,156.958
C02523=1040.563,-11.692,419.163,169.308,36.988,156.958
C02524=1040.569,-11.442,419.148,169.310,36.989,156.958
C02525=1040.575,-11.192,419.133,169.312,36.990,156.959
C02526=1040.581,-10.944,419.119,169.316,36.991,156.959
C02527=1040.588,-10.693,419.105,169.318,36.991,156.959
C02528=1040.594,-10.444,419.090,169.320,36.992,156.959
C02529=1040.600,-10.195,419.076,169.322,36.993,156.959
C02530=1040.607,-9.945,419.062,169.324,36.993,156.959
C02531=1040.613,-9.695,419.047,169.326,36.994,156.959
C02532=1040.619,-9.447,419.033,169.328,36.994,156.959
C02533=1040.626,-9.196,419.019,169.330,36.995,156.960
C02534=1040.632,-8.947,419.004,169.332,36.996,156.960
C02535=1040.638,-8.698,418.989,169.334,36.996,156.960
C02536=1040.645,-8.448,418.975,169.336,36.997,156.960
C02537=1040.651,-8.198,418.961,169.338,36.997,156.960
C02538=1040.657,-7.949,418.946,169.340,36.998,156.960
C02539=1040.664,-7.700,418.932,169.343,36.999,156.960
C02540=1040.670,-7.450,418.917,169.345,36.999,156.960
C02541=1040.676,-7.201,418.903,169.347,37.000,156.961
C02542=1040.683,-6.951,418.889,169.349,37.001,156.961
C02543=1040.689,-6.702,418.874,169.351,37.001,156.961
C02544=1040.696,-6.452,418.859,169.353,37.002,156.961
C02545=1040.701,-6.203,418.844,169.355,37.002,156.961
C02546=1040.708,-5.953,418.830,169.357,37.004,156.961
C02547=1040.715,-5.703,418.816,169.359,37.004,156.961
C02548=1040.721,-5.454,418.801,169.361,37.005,156.961
C02549=1040.727,-5.205,418.787,169.363,37.006,156.962
C02550=1040.734,-4.955,418.772,169.366,37.006,156.962
C02551=1040.740,-4.706,418.757,169.368,37.007,156.962
C02552=1040.746,-4.455,418.742,169.370,37.007,156.962
C02553=1040.753,-4.207,418.729,169.372,37.008,156.962
C02554=1040.759,-3.957,418.714,169.374,37.009,156.962
C02555=1040.766,-3.674,418.697,169.377,37.009,156.962
C02556=1040.774,-3.391,418.680,169.379,37.010,156.962
C02557=1040.781,-3.107,418.663,169.381,37.011,156.963
C02558=1040.788,-2.823,418.646,169.383,37.012,156.963
C02559=1040.793,-2.574,418.632,169.385,37.012,156.963
C02560=1040.800,-2.324,418.617,169.388,37.014,156.963
C02561=1040.806,-2.075,418.602,169.390,37.014,156.963
C02562=1040.813,-1.825,418.587,169.392,37.015,156.963
C02563=1040.818,-1.576,418.572,169.394,37.015,156.964
C02564=1040.825,-1.326,418.558,169.396,37.017,156.964
C02565=1040.831,-1.077,418.543,169.398,37.017,156.964
C02566=1040.838,-0.828,418.527,169.400,37.018,156.964
C02567=1040.844,-0.579,418.512,169.402,37.018,156.964
C02568=1040.850,-0.329,418.497,169.404,37.020,156.964
C02569=1040.856,-0.079,418.482,169.406,37.020,156.965
C02570=1040.863,0.170,418.468,169.409,37.021,156.965
C02571=1040.869,0.420,418.453,169.411,37.022,156.965
C02572=1040.875,0.669,418.438,169.413,37.023,156.965
C02573=1040.881,0.919,418.423,169.415,37.023,156.965
C02574=1040.888,1.168,418.408,169.417,37.024,156.965
C02575=1040.894,1.418,418.393,169.419,37.025,156.965
C02576=1040.900,1.668,418.378,169.421,37.025,156.966
C02577=1040.905,1.917,418.363,169.422,37.027,156.966
C02578=1040.912,2.166,418.347,169.424,37.027,156.966
C02579=1040.919,2.416,418.332,169.426,37.028,156.966
C02580=1040.925,2.665,418.317,169.429,37.028,156.966
C02581=1040.931,2.915,418.303,169.431,37.030,156.966
C02582=1040.938,3.165,418.288,169.433,37.030,156.967
C02583=1040.944,3.413,418.273,169.435,37.031,156.967
C02584=1040.950,3.663,418.258,169.437,37.031,156.967
C02585=1040.957,3.912,418.242,169.439,37.033,156.967
C02586=1040.963,4.162,418.227,169.441,37.033,156.967
C02587=1040.969,4.411,418.212,169.443,37.034,156.967
C02588=1040.976,4.661,418.198,169.445,37.035,156.967
C02589=1040.982,4.911,418.183,169.447,37.035,156.967
C02590=1040.989,5.160,418.167,169.450,37.036,156.968
C02591=1040.994,5.409,418.152,169.452,37.037,156.968
C02592=1041.000,5.659,418.137,169.454,37.038,156.968
C02593=1041.007,5.908,418.122,169.456,37.038,156.968
C02594=1041.013,6.157,418.106,169.458,37.040,156.968
C02595=1041.020,6.407,418.091,169.459,37.040,156.968
C02596=1041.026,6.657,418.076,169.461,37.041,156.969
C02597=1041.032,6.906,418.061,169.463,37.041,156.969
C02598=1041.039,7.155,418.046,169.465,37.042,156.969
C02599=1041.046,7.405,418.031,169.467,37.043,156.969
C02600=1041.052,7.655,418.016,169.470,37.044,156.969
C02601=1041.059,7.904,418.000,169.472,37.044,156.969
C02602=1041.064,8.154,417.985,169.474,37.045,156.969
C02603=1041.070,8.403,417.970,169.476,37.046,156.970
C02604=1041.077,8.652,417.954,169.478,37.047,156.970
C02605=1041.083,8.901,417.939,169.480,37.048,156.970
C02606=1041.089,9.151,417.924,169.482,37.048,156.970
C02607=1041.096,9.400,417.909,169.484,37.049,156.970
C02608=1041.103,9.650,417.894,169.486,37.050,156.970
C02609=1041.109,9.899,417.879,169.488,37.051,156.971
C02610=1041.116,10.148,417.863,169.491,37.051,156.971
C02611=1041.121,10.398,417.848,169.492,37.052,156.971
C02612=1041.128,10.648,417.833,169.494,37.052,156.971
C02613=1041.134,10.897,417.817,169.496,37.054,156.971
C02614=1041.141,11.147,417.802,169.498,37.054,156.971
C02615=1041.147,11.396,417.787,169.500,37.055,156.971
C02616=1041.154,11.645,417.772,169.502,37.056,156.972
C02617=1041.160,11.895,417.757,169.504,37.056,156.972
C02618=1041.167,12.144,417.741,169.506,37.057,156.972
C02619=1041.174,12.429,417.723,169.508,37.058,156.972
C02620=1041.181,12.716,417.706,169.511,37.059,156.972
C02621=1041.188,13.001,417.688,169.514,37.060,156.972
C02622=1041.196,13.286,417.670,169.516,37.060,156.973
C02623=1041.202,13.536,417.655,169.518,37.061,156.973
C02624=1041.209,13.785,417.640,169.520,37.062,156.973
C02625=1041.215,14.034,417.625,169.522,37.063,156.973
C02626=1041.221,14.284,417.609,169.523,37.064,156.973
C02627=1041.228,14.533,417.593,169.525,37.064,156.973
C02628=1041.234,14.782,417.578,169.527,37.065,156.974
C02629=1041.240,15.032,417.562,169.530,37.066,156.974
C02630=1041.247,15.281,417.547,169.532,37.067,156.974
C02631=1041.253,15.530,417.531,169.534,37.068,156.974
C02632=1041.260,15.781,417.515,169.536,37.068,156.974
C02633=1041.266,16.030,417.500,169.538,37.069,156.974
C02634=1041.272,16.279,417.483,169.539,37.070,156.974
C02635=1041.279,16.529,417.468,169.541,37.071,156.975
C02636=1041.285,16.778,417.453,169.543,37.072,156.975
C02637=1041.291,17.028,417.437,169.545,37.073,156.975
C02638=1041.298,17.277,417.421,169.548,37.073,156.975
C02639=1041.304,17.526,417.405,169.550,37.074,156.975
C02640=1041.310,17.776,417.390,169.552,37.075,156.975
C02641=1041.317,18.025,417.375,169.554,37.076,156.976
C02642=1041.323,18.275,417.358,169.556,37.076,156.976
C02643=1041.329,18.524,417.343,169.557,37.078,156.976
C02644=1041.335,18.774,417.327,169.559,37.078,156.976
C02645=1041.342,19.023,417.311,169.561,37.079,156.976
C02646=1041.349,19.273,417.296,169.563,37.080,156.976
C02647=1041.355,19.522,417.280,169.566,37.081,156.977
C02648=1041.361,19.771,417.264,169.568,37.081,156.977
C02649=1041.367,20.021,417.248,169.570,37.083,156.977
C02650=1041.374,20.270,417.233,169.572,37.083,156.977
C02651=1041.380,20.520,417.217,169.573,37.085,156.977
C02652=1041.386,20.769,417.201,169.575,37.085,156.977
C02653=1041.392,21.018,417.185,169.577,37.086,156.978
C02654=1041.399,21.268,417.170,169.579,37.087,156.978
C02655=1041.405,21.518,417.153,169.581,37.088,156.978
C02656=1041.412,21.767,417.138,169.584,37.089,156.978
C02657=1041.418,22.016,417.121,169.586,37.089,156.978
C02658=1041.425,22.265,417.106,169.587,37.090,156.978
C02659=1041.430,22.515,417.090,169.589,37.091,156.979
C02660=1041.437,22.764,417.075,169.591,37.092,156.979
C02661=1041.443,23.014,417.058,169.593,37.093,156.979
C02662=1041.449,23.263,417.042,169.595,37.094,156.979
C02663=1041.456,23.513,417.026,169.597,37.094,156.979
C02664=1041.462,23.762,417.010,169.600,37.096,156.980
C02665=1041.468,24.012,416.995,169.601,37.096,156.980
C02666=1041.474,24.261,416.979,169.603,37.098,156.980
C02667=1041.481,24.510,416.963,169.605,37.098,156.980
C02668=1041.487,24.759,416.947,169.607,37.099,156.980
C02669=1041.494,25.009,416.931,169.609,37.100,156.980
C02670=1041.500,25.258,416.914,169.611,37.101,156.981
C02671=1041.506,25.508,416.898,169.612,37.101,156.981
C02672=1041.513,25.757,416.882,169.615,37.102,156.981
C02673=1041.519,26.006,416.866,169.617,37.103,156.981
C02674=1041.526,26.256,416.850,169.619,37.104,156.981
C02675=1041.532,26.505,416.834,169.621,37.105,156.981
C02676=1041.538,26.755,416.818,169.623,37.105,156.982
C02677=1041.544,27.004,416.803,169.625,37.107,156.982
C02678=1041.550,27.254,416.786,169.626,37.107,156.982
C02679=1041.558,27.503,416.770,169.628,37.109,156.982
C02680=1041.564,27.753,416.754,169.630,37.109,156.982
C02681=1041.570,28.002,416.738,169.633,37.110,156.982
C02682=1041.576,28.251,416.722,169.635,37.111,156.983
C02683=1041.584,28.538,416.703,169.637,37.112,156.983
C02684=1041.591,28.825,416.684,169.639,37.113,156.983
C02685=1041.598,29.111,416.666,169.641,37.114,156.983
C02686=1041.605,29.398,416.647,169.643,37.115,156.983
C02687=1041.611,29.647,416.631,169.645,37.116,156.984
C02688=1041.618,29.897,416.614,169.648,37.117,156.984
C02689=1041.624,30.146,416.598,169.650,37.118,156.984
C02690=1041.630,30.396,416.582,169.651,37.119,156.984
C02691=1041.637,30.644,416.566,169.653,37.120,156.984
C02692=1041.643,30.894,416.549,169.655,37.121,156.985
C02693=1041.649,31.144,416.533,169.657,37.122,156.985
C02694=1041.655,31.393,416.516,169.659,37.122,156.985
C02695=1041.661,31.642,416.500,169.660,37.123,156.985
C02696=1041.668,31.892,416.484,169.662,37.124,156.985
C02697=1041.674,32.141,416.468,169.665,37.125,156.985
C02698=1041.681,32.390,416.451,169.667,37.126,156.986
C02699=1041.687,32.640,416.435,169.669,37.127,156.986
C02700=1041.693,32.890,416.418,169.671,37.128,156.986
C02701=1041.700,33.139,416.402,169.672,37.129,156.986
C02702=1041.706,33.388,416.386,169.674,37.130,156.986
C02703=1041.712,33.638,416.370,169.676,37.131,156.987
C02704=1041.719,33.887,416.353,169.678,37.131,156.987
C02705=1041.725,34.136,416.336,169.681,37.133,156.987
C02706=1041.731,34.385,416.321,169.682,37.133,156.987
C02707=1041.738,34.635,416.304,169.684,37.134,156.987
C02708=1041.744,34.885,416.288,169.686,37.135,156.987
C02709=1041.750,35.133,416.271,169.688,37.136,156.988
C02710=1041.757,35.383,416.254,169.690,37.137,156.988
C02711=1041.763,35.632,416.239,169.691,37.138,156.988
C02712=1041.769,35.882,416.222,169.693,37.139,156.988
C02713=1041.776,36.131,416.205,169.696,37.139,156.988
C02714=1041.782,36.380,416.189,169.698,37.141,156.989
C02715=1041.789,36.631,416.172,169.700,37.141,156.989
C02716=1041.795,36.879,416.155,169.702,37.142,156.989
C02717=1041.802,37.128,416.139,169.703,37.143,156.989
C02718=1041.808,37.378,416.123,169.705,37.144,156.989
C02719=1041.814,37.628,416.107,169.707,37.145,156.989
C02720=1041.820,37.876,416.090,169.710,37.146,156.990
C02721=1041.827,38.126,416.073,169.712,37.147,156.990
C02722=1041.833,38.375,416.056,169.713,37.148,156.990
C02723=1041.839,38.625,416.040,169.715,37.149,156.990
C02724=1041.846,38.875,416.023,169.717,37.150,156.990
C02725=1041.851,39.124,416.006,169.719,37.150,156.991
C02726=1041.857,39.373,415.989,169.720,37.152,156.991
C02727=1041.864,39.622,415.972,169.722,37.153,156.991
C02728=1041.870,39.872,415.956,169.725,37.154,156.991
C02729=1041.876,40.122,415.939,169.727,37.155,156.991
C02730=1041.883,40.371,415.922,169.729,37.155,156.991
C02731=1041.889,40.620,415.906,169.730,37.157,156.992
C02732=1041.896,40.869,415.888,169.732,37.157,156.992
C02733=1041.901,41.119,415.872,169.734,37.158,156.992
C02734=1041.908,41.367,415.855,169.736,37.159,156.992
C02735=1041.914,41.617,415.839,169.737,37.160,156.992
C02736=1041.921,41.866,415.822,169.740,37.162,156.993
C02737=1041.927,42.116,415.805,169.742,37.162,156.993
C02738=1041.933,42.365,415.788,169.744,37.163,156.993
C02739=1041.940,42.615,415.771,169.746,37.164,156.993
C02740=1041.946,42.864,415.754,169.747,37.165,156.993
C02741=1041.952,43.113,415.738,169.749,37.166,156.994
C02742=1041.959,43.362,415.721,169.751,37.167,156.994
C02743=1041.964,43.612,415.704,169.754,37.168,156.994
C02744=1041.971,43.862,415.687,169.755,37.169,156.994
C02745=1041.977,44.111,415.670,169.757,37.170,156.994
C02746=1041.983,44.360,415.653,169.759,37.171,156.995
C02747=1041.990,44.647,415.633,169.761,37.173,156.995
C02748=1041.997,44.933,415.614,169.763,37.173,156.995
C02749=1042.004,45.219,415.595,169.765,37.174,156.995
C02750=1042.011,45.507,415.575,169.768,37.176,156.996
C02751=1042.017,45.756,415.557,169.770,37.177,156.996
C02752=1042.024,46.005,415.540,169.771,37.178,156.996
C02753=1042.030,46.255,415.524,169.773,37.179,156.996
C02754=1042.036,46.504,415.506,169.775,37.180,156.996
C02755=1042.042,46.753,415.489,169.777,37.181,156.997
C02756=1042.048,47.002,415.473,169.778,37.182,156.997
C02757=1042.055,47.252,415.455,169.781,37.183,156.997
C02758=1042.060,47.501,415.438,169.783,37.184,156.997
C02759=1042.067,47.751,415.421,169.785,37.185,156.997
C02760=1042.073,48.000,415.404,169.786,37.186,156.998
C02761=1042.079,48.249,415.386,169.788,37.187,156.998
C02762=1042.086,48.498,415.369,169.790,37.188,156.998
C02763=1042.092,48.748,415.353,169.792,37.189,156.998
C02764=1042.098,48.997,415.335,169.794,37.190,156.999
C02765=1042.105,49.247,415.318,169.796,37.191,156.999
C02766=1042.111,49.495,415.301,169.798,37.192,156.999
C02767=1042.117,49.746,415.284,169.800,37.193,156.999
C02768=1042.123,49.994,415.267,169.801,37.194,156.999
C02769=1042.130,50.244,415.249,169.803,37.195,157.000
C02770=1042.135,50.493,415.232,169.805,37.196,157.000
C02771=1042.142,50.743,415.215,169.808,37.197,157.000
C02772=1042.147,50.992,415.198,169.809,37.198,157.000
C02773=1042.154,51.241,415.180,169.811,37.199,157.000
C02774=1042.160,51.490,415.163,169.813,37.200,157.001
C02775=1042.167,51.740,415.145,169.815,37.202,157.001
C02776=1042.173,51.989,415.128,169.816,37.202,157.001
C02777=1042.179,52.239,415.112,169.818,37.203,157.001
C02778=1042.185,52.488,415.094,169.821,37.204,157.001
C02779=1042.192,52.737,415.077,169.823,37.205,157.002
C02780=1042.198,52.986,415.060,169.824,37.206,157.002
C02781=1042.204,53.236,415.042,169.826,37.207,157.002
C02782=1042.211,53.485,415.025,169.828,37.208,157.002
C02783=1042.217,53.734,415.008,169.830,37.210,157.002
C02784=1042.223,53.984,414.990,169.832,37.210,157.003
C02785=1042.229,54.233,414.973,169.834,37.211,157.003
C02786=1042.235,54.483,414.955,169.836,37.212,157.003
C02787=1042.242,54.732,414.938,169.838,37.213,157.003
C02788=1042.249,54.981,414.921,169.840,37.214,157.003
C02789=1042.255,55.230,414.903,169.841,37.215,157.003
C02790=1042.261,55.479,414.886,169.843,37.216,157.004
C02791=1042.268,55.729,414.869,169.845,37.217,157.004
C02792=1042.274,55.978,414.851,169.848,37.218,157.004
C02793=1042.280,56.227,414.834,169.849,37.219,157.004
C02794=1042.286,56.477,414.816,169.851,37.220,157.004
C02795=1042.293,56.726,414.799,169.853,37.221,157.005
C02796=1042.299,56.975,414.782,169.855,37.222,157.005
C02797=1042.305,57.225,414.764,169.856,37.223,157.005
C02798=1042.312,57.473,414.747,169.858,37.224,157.005
C02799=1042.318,57.723,414.729,169.861,37.225,157.005
C02800=1042.325,57.973,414.712,169.863,37.226,157.006
C02801=1042.331,58.221,414.695,169.864,37.227,157.006
C02802=1042.337,58.471,414.677,169.866,37.228,157.006
C02803=1042.344,58.721,414.659,169.868,37.229,157.006
C02804=1042.349,58.970,414.642,169.870,37.230,157.006
C02805=1042.356,59.219,414.624,169.871,37.231,157.007
C02806=1042.363,59.468,414.607,169.873,37.232,157.007
C02807=1042.369,59.717,414.590,169.876,37.233,157.007
C02808=1042.376,59.967,414.572,169.878,37.233,157.007
C02809=1042.382,60.217,414.554,169.879,37.235,157.007
C02810=1042.388,60.465,414.537,169.881,37.236,157.008
C02811=1042.396,60.752,414.517,169.883,37.236,157.008
C02812=1042.402,61.038,414.497,169.885,37.238,157.008
C02813=1042.410,61.325,414.477,169.888,37.239,157.008
C02814=1042.418,61.611,414.456,169.890,37.240,157.009
C02815=1042.424,61.860,414.439,169.892,37.241,157.009
C02816=1042.430,62.110,414.421,169.894,37.242,157.009
C02817=1042.437,62.358,414.403,169.896,37.243,157.009
C02818=1042.443,62.607,414.386,169.897,37.244,157.009
C02819=1042.450,62.857,414.369,169.899,37.245,157.010
C02820=1042.456,63.106,414.351,169.901,37.246,157.010
C02821=1042.463,63.356,414.333,169.904,37.247,157.010
C02822=1042.469,63.605,414.316,169.905,37.247,157.010
C02823=1042.475,63.855,414.298,169.907,37.249,157.010
C02824=1042.482,64.103,414.280,169.909,37.249,157.010
C02825=1042.488,64.353,414.262,169.911,37.250,157.011
C02826=1042.494,64.602,414.245,169.912,37.252,157.011
C02827=1042.501,64.852,414.227,169.915,37.253,157.011
C02828=1042.507,65.101,414.209,169.917,37.254,157.011
C02829=1042.513,65.350,414.191,169.919,37.255,157.012
C02830=1042.519,65.599,414.174,169.920,37.256,157.012
C02831=1042.525,65.849,414.156,169.922,37.257,157.012
C02832=1042.532,66.098,414.137,169.924,37.258,157.012
C02833=1042.539,66.348,414.120,169.925,37.259,157.012
C02834=1042.544,66.597,414.102,169.928,37.260,157.013
C02835=1042.551,66.846,414.084,169.930,37.261,157.013
C02836=1042.557,67.095,414.066,169.932,37.262,157.013
C02837=1042.564,67.345,414.048,169.933,37.263,157.013
C02838=1042.570,67.593,414.030,169.935,37.264,157.013
C02839=1042.576,67.843,414.012,169.937,37.265,157.014
C02840=1042.582,68.093,413.994,169.939,37.266,157.014
C02841=1042.589,68.342,413.976,169.941,37.267,157.014
C02842=1042.594,68.591,413.959,169.943,37.268,157.014
C02843=1042.601,68.840,413.940,169.945,37.269,157.015
C02844=1042.607,69.089,413.922,169.947,37.270,157.015
C02845=1042.614,69.339,413.905,169.948,37.271,157.015
C02846=1042.620,69.588,413.886,169.950,37.272,157.015
C02847=1042.626,69.837,413.869,169.953,37.274,157.015
C02848=1042.632,70.086,413.850,169.954,37.274,157.016
C02849=1042.638,70.336,413.832,169.956,37.276,157.016
C02850=1042.645,70.585,413.813,169.958,37.277,157.016
C02851=1042.651,70.834,413.796,169.960,37.278,157.016
C02852=1042.657,71.084,413.778,169.961,37.279,157.016
C02853=1042.664,71.333,413.760,169.963,37.280,157.017
C02854=1042.670,71.582,413.742,169.966,37.281,157.017
C02855=1042.676,71.831,413.723,169.968,37.282,157.017
C02856=1042.682,72.081,413.706,169.969,37.283,157.017
C02857=1042.688,72.330,413.687,169.971,37.284,157.018
C02858=1042.694,72.579,413.669,169.973,37.285,157.018
C02859=1042.701,72.829,413.650,169.974,37.287,157.018
C02860=1042.707,73.078,413.632,169.976,37.287,157.018
C02861=1042.714,73.327,413.614,169.979,37.288,157.018
C02862=1042.720,73.575,413.596,169.981,37.290,157.019
C02863=1042.726,73.825,413.578,169.982,37.291,157.019
C02864=1042.732,74.074,413.560,169.984,37.291,157.019
C02865=1042.738,74.324,413.542,169.986,37.293,157.019
C02866=1042.745,74.573,413.523,169.987,37.294,157.020
C02867=1042.751,74.822,413.504,169.990,37.295,157.020
C02868=1042.757,75.072,413.486,169.992,37.296,157.020
C02869=1042.763,75.320,413.468,169.994,37.297,157.020
C02870=1042.769,75.570,413.450,169.995,37.298,157.020
C02871=1042.776,75.819,413.432,169.997,37.299,157.021
C02872=1042.782,76.068,413.413,169.999,37.300,157.021
C02873=1042.788,76.318,413.395,170.002,37.301,157.021
C02874=1042.795,76.567,413.376,170.003,37.302,157.021
C02875=1042.802,76.853,413.356,170.005,37.304,157.022
C02876=1042.809,77.140,413.335,170.007,37.305,157.022
C02877=1042.817,77.426,413.314,170.009,37.306,157.022
C02878=1042.823,77.711,413.292,170.011,37.307,157.022
C02879=1042.830,77.960,413.274,170.013,37.308,157.022
C02880=1042.836,78.210,413.256,170.016,37.309,157.023
C02881=1042.842,78.459,413.237,170.017,37.310,157.023
C02882=1042.849,78.708,413.219,170.019,37.312,157.023
C02883=1042.855,78.957,413.200,170.021,37.313,157.023
C02884=1042.861,79.207,413.182,170.023,37.314,157.024
C02885=1042.867,79.457,413.163,170.024,37.315,157.024
C02886=1042.873,79.705,413.144,170.027,37.316,157.024
C02887=1042.879,79.954,413.126,170.029,37.317,157.024
C02888=1042.885,80.203,413.107,170.030,37.318,157.025
C02889=1042.892,80.453,413.089,170.032,37.319,157.025
C02890=1042.897,80.702,413.070,170.034,37.321,157.025
C02891=1042.904,80.952,413.051,170.035,37.321,157.025
C02892=1042.910,81.201,413.033,170.038,37.323,157.025
C02893=1042.917,81.450,413.014,170.040,37.324,157.026
C02894=1042.923,81.699,412.995,170.042,37.325,157.026
C02895=1042.928,81.949,412.977,170.043,37.326,157.026
C02896=1042.935,82.198,412.958,170.045,37.327,157.026
C02897=1042.941,82.447,412.940,170.047,37.328,157.027
C02898=1042.947,82.696,412.921,170.049,37.329,157.027
C02899=1042.953,82.945,412.903,170.051,37.330,157.027
C02900=1042.959,83.194,412.883,170.053,37.332,157.027
C02901=1042.966,83.443,412.865,170.055,37.333,157.028
C02902=1042.972,83.692,412.846,170.056,37.334,157.028
C02903=1042.978,83.942,412.827,170.058,37.335,157.028
C02904=1042.985,84.191,412.809,170.061,37.336,157.028
C02905=1042.990,84.441,412.790,170.063,37.337,157.028
C02906=1042.997,84.690,412.772,170.064,37.338,157.029
C02907=1043.003,84.939,412.753,170.066,37.340,157.029
C02908=1043.010,85.188,412.734,170.068,37.340,157.029
C02909=1043.015,85.438,412.715,170.069,37.341,157.029
C02910=1043.022,85.687,412.696,170.072,37.343,157.030
C02911=1043.028,85.936,412.678,170.074,37.344,157.030
C02912=1043.035,86.185,412.659,170.076,37.345,157.030
C02913=1043.041,86.434,412.640,170.077,37.346,157.030
C02914=1043.047,86.684,412.621,170.079,37.347,157.030
C02915=1043.053,86.933,412.603,170.081,37.348,157.031
C02916=1043.059,87.182,412.584,170.084,37.349,157.031
C02917=1043.066,87.431,412.565,170.085,37.350,157.031
C02918=1043.072,87.680,412.546,170.087,37.351,157.031
C02919=1043.078,87.929,412.527,170.089,37.352,157.032
C02920=1043.084,88.179,412.509,170.091,37.354,157.032
C02921=1043.091,88.428,412.490,170.092,37.355,157.032
C02922=1043.097,88.677,412.471,170.094,37.355,157.032
C02923=1043.104,88.927,412.452,170.097,37.357,157.032
C02924=1043.110,89.176,412.433,170.098,37.358,157.033
C02925=1043.116,89.425,412.415,170.100,37.359,157.033
C02926=1043.122,89.675,412.395,170.102,37.360,157.033
C02927=1043.129,89.923,412.376,170.104,37.361,157.033
C02928=1043.135,90.172,412.357,170.105,37.362,157.034
C02929=1043.141,90.422,412.338,170.108,37.363,157.034
C02930=1043.147,90.671,412.319,170.110,37.364,157.034
C02931=1043.153,90.920,412.300,170.112,37.366,157.034
C02932=1043.160,91.169,412.281,170.113,37.367,157.035
C02933=1043.165,91.419,412.262,170.115,37.368,157.035
C02934=1043.172,91.667,412.243,170.117,37.369,157.035
C02935=1043.178,91.917,412.224,170.119,37.370,157.035
C02936=1043.184,92.166,412.205,170.121,37.371,157.036
C02937=1043.190,92.415,412.186,170.123,37.372,157.036
C02938=1043.196,92.664,412.166,170.125,37.374,157.036
C02939=1043.204,92.950,412.145,170.127,37.375,157.036
C02940=1043.211,93.236,412.123,170.130,37.376,157.037
C02941=1043.217,93.522,412.100,170.132,37.378,157.037
C02942=1043.225,93.809,412.079,170.134,37.379,157.037
C02943=1043.231,94.057,412.059,170.135,37.380,157.037
C02944=1043.237,94.307,412.040,170.137,37.382,157.038
C02945=1043.243,94.556,412.021,170.139,37.382,157.038
C02946=1043.249,94.805,412.002,170.141,37.383,157.038
C02947=1043.256,95.054,411.983,170.143,37.385,157.038
C02948=1043.262,95.304,411.963,170.145,37.386,157.039
C02949=1043.268,95.553,411.944,170.147,37.387,157.039
C02950=1043.275,95.802,411.924,170.148,37.388,157.039
C02951=1043.280,96.051,411.905,170.151,37.389,157.039
C02952=1043.287,96.300,411.887,170.153,37.391,157.040
C02953=1043.293,96.549,411.867,170.155,37.391,157.040
C02954=1043.299,96.798,411.848,170.156,37.392,157.040
C02955=1043.305,97.048,411.828,170.158,37.394,157.040
C02956=1043.312,97.297,411.809,170.160,37.395,157.040
C02957=1043.318,97.546,411.790,170.163,37.396,157.041
C02958=1043.324,97.795,411.771,170.164,37.397,157.041
C02959=1043.330,98.044,411.751,170.166,37.399,157.041
C02960=1043.337,98.293,411.733,170.168,37.400,157.041
C02961=1043.343,98.543,411.712,170.170,37.400,157.042
C02962=1043.349,98.792,411.693,170.171,37.402,157.042
C02963=1043.355,99.041,411.674,170.174,37.403,157.042
C02964=1043.361,99.290,411.654,170.176,37.404,157.042
C02965=1043.368,99.539,411.636,170.177,37.405,157.043
C02966=1043.374,99.789,411.615,170.179,37.406,157.043
C02967=1043.381,100.038,411.597,170.181,37.407,157.043
C02968=1043.387,100.287,411.577,170.183,37.408,157.043
C02969=1043.392,100.536,411.557,170.186,37.409,157.043
C02970=1043.399,100.785,411.538,170.187,37.411,157.044
C02971=1043.405,101.035,411.519,170.189,37.412,157.044
C02972=1043.411,101.284,411.499,170.191,37.413,157.044
C02973=1043.417,101.533,411.479,170.192,37.414,157.044
C02974=1043.423,101.782,411.459,170.194,37.415,157.045
C02975=1043.430,102.031,411.441,170.197,37.417,157.045
C02976=1043.436,102.280,411.421,170.199,37.418,157.045
C02977=1043.442,102.529,411.400,170.200,37.419,157.045
C02978=1043.448,102.779,411.381,170.202,37.420,157.046
C02979=1043.454,103.028,411.361,170.204,37.422,157.046
C02980=1043.460,103.277,411.342,170.207,37.423,157.046
C02981=1043.466,103.526,411.323,170.208,37.424,157.046
C02982=1043.473,103.775,411.302,170.210,37.425,157.047
C02983=1043.479,104.025,411.283,170.212,37.426,157.047
C02984=1043.485,104.273,411.263,170.213,37.428,157.047
C02985=1043.490,104.523,411.244,170.216,37.429,157.047
C02986=1043.498,104.772,411.224,170.218,37.430,157.048
C02987=1043.504,105.021,411.204,170.220,37.431,157.048
C02988=1043.509,105.270,411.185,170.221,37.432,157.048
C02989=1043.515,105.519,411.165,170.223,37.434,157.048
C02990=1043.522,105.769,411.145,170.225,37.435,157.049
C02991=1043.528,106.018,411.125,170.228,37.435,157.049
C02992=1043.534,106.267,411.106,170.229,37.437,157.049
C02993=1043.540,106.515,411.086,170.231,37.438,157.049
C02994=1043.547,106.765,411.066,170.233,37.439,157.050
C02995=1043.553,107.014,411.046,170.235,37.440,157.050
C02996=1043.559,107.263,411.027,170.237,37.441,157.050
C02997=1043.565,107.512,411.007,170.239,37.443,157.050
C02998=1043.572,107.762,410.988,170.241,37.444,157.051
C02999=1043.578,108.011,410.968,170.243,37.445,157.051
C03000=1043.584,108.259,410.948,170.245,37.446,157.051
C03001=1043.590,108.509,410.927,170.246,37.448,157.051
C03002=1043.596,108.758,410.908,170.249,37.449,157.052
C03003=1043.603,109.044,410.886,170.251,37.450,157.052
C03004=1043.610,109.330,410.863,170.253,37.451,157.052
C03005=1043.617,109.617,410.839,170.255,37.452,157.052
C03006=1043.625,109.902,410.816,170.257,37.454,157.053
C03007=1043.631,110.151,410.797,170.260,37.455,157.053
C03008=1043.637,110.400,410.777,170.262,37.457,157.053
C03009=1043.643,110.650,410.757,170.264,37.457,157.053
C03010=1043.649,110.898,410.737,170.265,37.458,157.054
C03011=1043.655,111.147,410.717,170.267,37.460,157.054
C03012=1043.662,111.397,410.697,170.269,37.461,157.054
C03013=1043.668,111.646,410.677,170.272,37.462,157.054
C03014=1043.674,111.895,410.657,170.273,37.463,157.055
C03015=1043.680,112.145,410.637,170.275,37.464,157.055
C03016=1043.686,112.393,410.617,170.277,37.466,157.055
C03017=1043.693,112.643,410.597,170.279,37.467,157.055
C03018=1043.699,112.892,410.577,170.281,37.468,157.056
C03019=1043.705,113.140,410.557,170.283,37.469,157.056
C03020=1043.711,113.390,410.537,170.285,37.470,157.056
C03021=1043.717,113.639,410.517,170.287,37.472,157.056
C03022=1043.723,113.888,410.497,170.288,37.473,157.057
C03023=1043.730,114.137,410.476,170.291,37.475,157.057
C03024=1043.735,114.386,410.456,170.293,37.476,157.057
C03025=1043.741,114.635,410.436,170.295,37.477,157.058
C03026=1043.748,114.885,410.416,170.296,37.478,157.058
C03027=1043.754,115.133,410.396,170.298,37.480,157.058
C03028=1043.759,115.383,410.375,170.300,37.481,157.058
C03029=1043.766,115.632,410.355,170.303,37.482,157.059
C03030=1043.772,115.881,410.335,170.304,37.483,157.059
C03031=1043.777,116.130,410.314,170.306,37.485,157.059
C03032=1043.783,116.379,410.294,170.308,37.486,157.060
C03033=1043.789,116.628,410.274,170.311,37.487,157.060
C03034=1043.796,116.876,410.253,170.313,37.489,157.060
C03035=1043.802,117.126,410.232,170.314,37.490,157.060
C03036=1043.808,117.375,410.212,170.316,37.491,157.061
C03037=1043.814,117.625,410.192,170.318,37.492,157.061
C03038=1043.819,117.874,410.171,170.320,37.493,157.061
C03039=1043.825,118.123,410.152,170.322,37.495,157.061
C03040=1043.832,118.372,410.131,170.324,37.496,157.062
C03041=1043.838,118.621,410.111,170.326,37.498,157.062
C03042=1043.844,118.870,410.090,170.328,37.499,157.062
C03043=1043.850,119.119,410.070,170.329,37.500,157.062
C03044=1043.856,119.368,410.050,170.332,37.501,157.063
C03045=1043.862,119.618,410.029,170.334,37.502,157.063
C03046=1043.868,119.866,410.009,170.336,37.504,157.063
C03047=1043.875,120.115,409.988,170.338,37.505,157.063
C03048=1043.880,120.364,409.967,170.339,37.506,157.064
C03049=1043.887,120.614,409.947,170.342,37.507,157.064
C03050=1043.893,120.863,409.927,170.344,37.509,157.064
C03051=1043.899,121.112,409.907,170.346,37.510,157.065
C03052=1043.905,121.361,409.885,170.348,37.511,157.065
C03053=1043.911,121.610,409.865,170.349,37.513,157.065
C03054=1043.917,121.859,409.845,170.352,37.514,157.065
C03055=1043.923,122.108,409.824,170.354,37.515,157.066
C03056=1043.930,122.357,409.803,170.356,37.516,157.066
C03057=1043.936,122.606,409.783,170.357,37.518,157.066
C03058=1043.942,122.856,409.763,170.359,37.519,157.066
C03059=1043.948,123.104,409.742,170.362,37.520,157.067
C03060=1043.954,123.353,409.722,170.364,37.521,157.067
C03061=1043.960,123.603,409.701,170.366,37.522,157.067
C03062=1043.967,123.851,409.680,170.368,37.523,157.067
C03063=1043.973,124.100,409.660,170.369,37.525,157.068
C03064=1043.978,124.350,409.639,170.372,37.527,157.068
C03065=1043.985,124.598,409.618,170.374,37.528,157.068
C03066=1043.991,124.848,409.598,170.376,37.529,157.069
C03067=1043.998,125.133,409.574,170.378,37.530,157.069
C03068=1044.006,125.420,409.551,170.380,37.531,157.069
C03069=1044.012,125.706,409.527,170.383,37.533,157.069
C03070=1044.019,125.992,409.503,170.385,37.534,157.070
C03071=1044.025,126.241,409.483,170.387,37.536,157.070
C03072=1044.032,126.489,409.462,170.389,37.537,157.070
C03073=1044.038,126.739,409.441,170.391,37.538,157.071
C03074=1044.045,126.987,409.420,170.393,37.539,157.071
C03075=1044.051,127.236,409.400,170.395,37.541,157.071
C03076=1044.056,127.486,409.379,170.397,37.542,157.071
C03077=1044.063,127.735,409.358,170.399,37.543,157.072
C03078=1044.069,127.984,409.338,170.401,37.545,157.072
C03079=1044.075,128.233,409.317,170.404,37.546,157.072
C03080=1044.081,128.482,409.297,170.405,37.547,157.072
C03081=1044.088,128.731,409.275,170.407,37.548,157.073
C03082=1044.094,128.981,409.255,170.409,37.549,157.073
C03083=1044.101,129.229,409.234,170.411,37.550,157.073
C03084=1044.106,129.479,409.213,170.414,37.552,157.073
C03085=1044.113,129.727,409.193,170.416,37.553,157.074
C03086=1044.119,129.976,409.172,170.418,37.554,157.074
C03087=1044.125,130.225,409.151,170.419,37.555,157.074
C03088=1044.131,130.474,409.131,170.421,37.556,157.074
C03089=1044.138,130.723,409.110,170.424,37.558,157.075
C03090=1044.144,130.973,409.089,170.426,37.559,157.075
C03091=1044.150,131.221,409.068,170.428,37.560,157.075
C03092=1044.157,131.470,409.046,170.430,37.562,157.076
C03093=1044.162,131.720,409.025,170.431,37.563,157.076
C03094=1044.169,131.968,409.005,170.434,37.564,157.076
C03095=1044.175,132.218,408.984,170.436,37.565,157.076
C03096=1044.181,132.467,408.962,170.438,37.567,157.077
C03097=1044.187,132.716,408.942,170.440,37.568,157.077
C03098=1044.193,132.965,408.921,170.442,37.570,157.077
C03099=1044.199,133.214,408.899,170.445,37.571,157.078
C03100=1044.205,133.463,408.878,170.446,37.572,157.078
C03101=1044.212,133.712,408.857,170.448,37.573,157.078
C03102=1044.217,133.961,408.836,170.450,37.574,157.078
C03103=1044.224,134.210,408.815,170.453,37.576,157.079
C03104=1044.230,134.459,408.793,170.455,37.577,157.079
C03105=1044.235,134.708,408.773,170.457,37.579,157.079
C03106=1044.242,134.957,408.752,170.458,37.580,157.079
C03107=1044.248,135.207,408.730,170.460,37.581,157.080
C03108=1044.254,135.455,408.709,170.463,37.583,157.080
C03109=1044.260,135.705,408.689,170.465,37.584,157.080
C03110=1044.267,135.954,408.667,170.467,37.585,157.081
C03111=1044.272,136.202,408.646,170.469,37.586,157.081
C03112=1044.279,136.451,408.625,170.471,37.588,157.081
C03113=1044.285,136.700,408.603,170.473,37.589,157.082
C03114=1044.290,136.949,408.582,170.475,37.591,157.082
C03115=1044.297,137.199,408.561,170.477,37.592,157.082
C03116=1044.303,137.448,408.540,170.479,37.593,157.082
C03117=1044.310,137.697,408.518,170.481,37.594,157.083
C03118=1044.315,137.945,408.497,170.484,37.596,157.083
C03119=1044.321,138.194,408.475,170.486,37.597,157.083
C03120=1044.328,138.443,408.454,170.488,37.598,157.083
C03121=1044.334,138.692,408.434,170.489,37.600,157.084
C03122=1044.340,138.942,408.412,170.491,37.601,157.084
C03123=1044.346,139.191,408.390,170.494,37.603,157.084
C03124=1044.353,139.440,408.369,170.496,37.604,157.085
C03125=1044.358,139.688,408.348,170.498,37.605,157.085
C03126=1044.364,139.938,408.326,170.500,37.606,157.085
C03127=1044.371,140.187,408.305,170.503,37.608,157.086
C03128=1044.376,140.435,408.284,170.505,37.609,157.086
C03129=1044.382,140.684,408.262,170.506,37.610,157.086
C03130=1044.389,140.934,408.240,170.508,37.612,157.086
C03131=1044.395,141.219,408.216,170.510,37.613,157.087
C03132=1044.403,141.505,408.191,170.514,37.615,157.087
C03133=1044.409,141.790,408.166,170.516,37.617,157.087
C03134=1044.416,142.076,408.142,170.518,37.618,157.088
C03135=1044.422,142.326,408.120,170.520,37.619,157.088
C03136=1044.428,142.575,408.098,170.523,37.621,157.088
C03137=1044.434,142.823,408.077,170.525,37.622,157.089
C03138=1044.440,143.072,408.056,170.526,37.624,157.089
C03139=1044.446,143.322,408.034,170.528,37.625,157.089
C03140=1044.453,143.571,408.013,170.531,37.627,157.089
C03141=1044.459,143.818,407.991,170.533,37.628,157.090
C03142=1044.465,144.068,407.969,170.535,37.629,157.090
C03143=1044.471,144.317,407.948,170.537,37.631,157.090
C03144=1044.478,144.566,407.926,170.539,37.632,157.091
C03145=1044.484,144.815,407.904,170.542,37.633,157.091
C03146=1044.489,145.064,407.883,170.544,37.635,157.091
C03147=1044.496,145.313,407.861,170.546,37.636,157.092
C03148=1044.502,145.562,407.840,170.548,37.637,157.092
C03149=1044.508,145.811,407.817,170.550,37.638,157.092
C03150=1044.514,146.060,407.796,170.552,37.640,157.092
C03151=1044.520,146.309,407.774,170.554,37.641,157.093
C03152=1044.527,146.558,407.753,170.556,37.643,157.093
C03153=1044.532,146.807,407.731,170.559,37.644,157.093
C03154=1044.538,147.056,407.710,170.561,37.646,157.094
C03155=1044.545,147.305,407.687,170.563,37.647,157.094
C03156=1044.551,147.554,407.666,170.565,37.649,157.094
C03157=1044.557,147.803,407.644,170.567,37.650,157.095
C03158=1044.563,148.052,407.622,170.570,37.651,157.095
C03159=1044.570,148.301,407.600,170.572,37.653,157.095
C03160=1044.575,148.549,407.579,170.574,37.654,157.095
C03161=1044.581,148.799,407.557,170.575,37.655,157.096
C03162=1044.587,149.047,407.534,170.578,37.657,157.096
C03163=1044.593,149.297,407.513,170.580,37.658,157.096
C03164=1044.600,149.546,407.491,170.582,37.660,157.097
C03165=1044.606,149.794,407.469,170.584,37.661,157.097
C03166=1044.612,150.044,407.447,170.586,37.662,157.097
C03167=1044.617,150.292,407.425,170.589,37.664,157.098
C03168=1044.624,150.541,407.403,170.591,37.665,157.098
C03169=1044.630,150.790,407.381,170.593,37.666,157.098
C03170=1044.636,151.039,407.359,170.595,37.668,157.099
C03171=1044.642,151.288,407.337,170.598,37.669,157.099
C03172=1044.648,151.538,407.315,170.600,37.671,157.099
C03173=1044.654,151.786,407.292,170.602,37.672,157.099
C03174=1044.660,152.035,407.271,170.604,37.674,157.100
C03175=1044.667,152.285,407.249,170.607,37.675,157.100
C03176=1044.672,152.533,407.226,170.609,37.677,157.100
C03177=1044.678,152.783,407.205,170.610,37.678,157.101
C03178=1044.684,153.031,407.183,170.612,37.680,157.101
C03179=1044.690,153.280,407.161,170.615,37.681,157.101
C03180=1044.697,153.528,407.139,170.617,37.683,157.102
C03181=1044.702,153.778,407.116,170.619,37.684,157.102
C03182=1044.709,154.026,407.094,170.621,37.686,157.102
C03183=1044.715,154.276,407.072,170.623,37.687,157.103
C03184=1044.721,154.524,407.050,170.626,37.688,157.103
C03185=1044.727,154.774,407.028,170.628,37.690,157.103
C03186=1044.733,155.022,407.006,170.630,37.691,157.103
C03187=1044.739,155.272,406.984,170.632,37.693,157.104
C03188=1044.745,155.520,406.961,170.635,37.694,157.104
C03189=1044.751,155.770,406.939,170.637,37.696,157.104
C03190=1044.757,156.019,406.916,170.639,37.697,157.105
C03191=1044.764,156.267,406.894,170.641,37.699,157.105
C03192=1044.770,156.516,406.872,170.644,37.700,157.105
C03193=1044.775,156.765,406.849,170.646,37.702,157.106
C03194=1044.782,157.014,406.828,170.648,37.703,157.106
C03195=1044.789,157.299,406.802,170.650,37.705,157.106
C03196=1044.796,157.585,406.777,170.653,37.706,157.107
C03197=1044.803,157.870,406.751,170.656,37.708,157.107
C03198=1044.809,158.155,406.725,170.658,37.710,157.108
C03199=1044.815,158.404,406.703,170.661,37.711,157.108
C03200=1044.822,158.652,406.680,170.663,37.713,157.108
C03201=1044.827,158.902,406.658,170.665,37.714,157.108
C03202=1044.834,159.151,406.636,170.667,37.715,157.109
C03203=1044.840,159.400,406.613,170.670,37.717,157.109
C03204=1044.846,159.649,406.591,170.672,37.718,157.109
C03205=1044.853,159.898,406.569,170.674,37.720,157.110
C03206=1044.859,160.147,406.546,170.676,37.721,157.110
C03207=1044.865,160.395,406.523,170.679,37.723,157.110
C03208=1044.870,160.645,406.501,170.681,37.725,157.111
C03209=1044.876,160.894,406.478,170.683,37.726,157.111
C03210=1044.883,161.142,406.456,170.685,37.728,157.111
C03211=1044.888,161.391,406.433,170.688,37.729,157.112
C03212=1044.894,161.640,406.410,170.690,37.731,157.112
C03213=1044.900,161.889,406.387,170.692,37.732,157.113
C03214=1044.905,162.139,406.365,170.694,37.734,157.113
C03215=1044.912,162.387,406.342,170.697,37.735,157.113
C03216=1044.917,162.636,406.319,170.699,37.737,157.114
C03217=1044.923,162.885,406.296,170.701,37.739,157.114
C03218=1044.929,163.134,406.274,170.703,37.740,157.114
C03219=1044.935,163.382,406.251,170.706,37.742,157.115
C03220=1044.941,163.631,406.228,170.708,37.744,157.115
C03221=1044.947,163.880,406.205,170.710,37.745,157.115
C03222=1044.953,164.129,406.182,170.713,37.747,157.116
C03223=1044.958,164.378,406.159,170.715,37.748,157.116
C03224=1044.965,164.627,406.137,170.717,37.750,157.116
C03225=1044.971,164.876,406.114,170.719,37.751,157.117
C03226=1044.976,165.124,406.091,170.722,37.753,157.117
C03227=1044.982,165.373,406.068,170.724,37.755,157.117
C03228=1044.988,165.622,406.045,170.726,37.756,157.118
C03229=1044.995,165.872,406.023,170.728,37.758,157.118
C03230=1045.001,166.120,406.000,170.731,37.760,157.118
C03231=1045.006,166.369,405.977,170.733,37.761,157.119
C03232=1045.012,166.618,405.954,170.735,37.763,157.119
C03233=1045.018,166.867,405.931,170.738,37.765,157.120
C03234=1045.023,167.116,405.908,170.740,37.766,157.120
C03235=1045.030,167.365,405.885,170.742,37.767,157.120
C03236=1045.036,167.613,405.863,170.744,37.769,157.121
C03237=1045.042,167.862,405.839,170.747,37.771,157.121
C03238=1045.048,168.111,405.816,170.749,37.772,157.121
C03239=1045.054,168.360,405.793,170.751,37.774,157.122
C03240=1045.060,168.609,405.770,170.753,37.776,157.122
C03241=1045.066,168.858,405.747,170.756,37.778,157.122
C03242=1045.072,169.107,405.724,170.758,37.779,157.123
C03243=1045.077,169.356,405.701,170.760,37.781,157.123
C03244=1045.084,169.605,405.677,170.763,37.782,157.123
C03245=1045.090,169.853,405.654,170.765,37.783,157.124
C03246=1045.096,170.102,405.632,170.768,37.785,157.124
C03247=1045.102,170.351,405.609,170.770,37.787,157.124
C03248=1045.108,170.600,405.586,170.773,37.788,157.125
C03249=1045.114,170.848,405.563,170.775,37.790,157.125
C03250=1045.120,171.098,405.539,170.777,37.792,157.126
C03251=1045.126,171.347,405.516,170.779,37.794,157.126
C03252=1045.132,171.595,405.493,170.782,37.795,157.126
C03253=1045.138,171.843,405.470,170.784,37.797,157.127
C03254=1045.145,172.093,405.447,170.786,37.798,157.127
C03255=1045.150,172.342,405.424,170.789,37.800,157.127
C03256=1045.156,172.591,405.401,170.791,37.801,157.128
C03257=1045.162,172.839,405.377,170.793,37.803,157.128
C03258=1045.168,173.089,405.354,170.796,37.805,157.128
C03259=1045.175,173.373,405.328,170.799,37.807,157.129
C03260=1045.182,173.658,405.301,170.801,37.808,157.129
C03261=1045.190,173.943,405.275,170.804,37.810,157.130
C03262=1045.196,174.227,405.248,170.807,37.812,157.130
C03263=1045.203,174.477,405.225,170.809,37.814,157.130
C03264=1045.208,174.726,405.202,170.811,37.815,157.131
C03265=1045.214,174.974,405.178,170.813,37.817,157.131
C03266=1045.220,175.223,405.155,170.817,37.818,157.131
C03267=1045.227,175.472,405.132,170.819,37.820,157.132
C03268=1045.233,175.721,405.109,170.821,37.822,157.132
C03269=1045.239,175.969,405.086,170.824,37.823,157.132
C03270=1045.246,176.218,405.062,170.826,37.825,157.133
C03271=1045.251,176.467,405.039,170.828,37.827,157.133
C03272=1045.257,176.716,405.015,170.830,37.828,157.134
C03273=1045.264,176.965,404.992,170.834,37.830,157.134
C03274=1045.269,177.214,404.969,170.836,37.831,157.134
C03275=1045.276,177.463,404.945,170.838,37.833,157.135
C03276=1045.283,177.712,404.923,170.841,37.835,157.135
C03277=1045.289,177.960,404.899,170.843,37.836,157.135
C03278=1045.295,178.210,404.876,170.845,37.838,157.136
C03279=1045.301,178.458,404.852,170.847,37.840,157.136
C03280=1045.307,178.707,404.829,170.851,37.841,157.137
C03281=1045.313,178.956,404.805,170.853,37.842,157.137
C03282=1045.319,179.204,404.781,170.855,37.844,157.137
C03283=1045.326,179.454,404.758,170.858,37.846,157.138
C03284=1045.332,179.702,404.734,170.860,37.848,157.138
C03285=1045.337,179.951,404.711,170.862,37.849,157.138
C03286=1045.344,180.200,404.687,170.865,37.851,157.139
C03287=1045.350,180.449,404.664,170.868,37.853,157.139
C03288=1045.357,180.697,404.641,170.870,37.854,157.139
C03289=1045.363,180.946,404.617,170.872,37.856,157.140
C03290=1045.370,181.195,404.594,170.874,37.857,157.140
C03291=1045.376,181.443,404.570,170.878,37.859,157.140
C03292=1045.382,181.693,404.547,170.880,37.861,157.141
C03293=1045.388,181.941,404.523,170.882,37.863,157.141
C03294=1045.395,182.190,404.499,170.885,37.864,157.142
C03295=1045.400,182.439,404.476,170.887,37.865,157.142
C03296=1045.407,182.688,404.452,170.890,37.867,157.142
C03297=1045.413,182.936,404.429,170.893,37.869,157.143
C03298=1045.419,183.186,404.405,170.895,37.871,157.143
C03299=1045.425,183.434,404.382,170.897,37.872,157.143
C03300=1045.432,183.683,404.358,170.899,37.874,157.144
C03301=1045.438,183.932,404.334,170.903,37.875,157.144
C03302=1045.445,184.181,404.310,170.905,37.877,157.145
C03303=1045.450,184.430,404.286,170.907,37.879,157.145
C03304=1045.456,184.678,404.263,170.910,37.881,157.145
C03305=1045.462,184.927,404.238,170.912,37.883,157.146
C03306=1045.468,185.176,404.214,170.914,37.885,157.146
C03307=1045.474,185.425,404.190,170.918,37.887,157.147
C03308=1045.480,185.673,404.166,170.920,37.888,157.147
C03309=1045.485,185.922,404.142,170.922,37.890,157.147
C03310=1045.492,186.171,404.118,170.925,37.892,157.148
C03311=1045.497,186.419,404.094,170.927,37.894,157.148
C03312=1045.504,186.668,404.070,170.930,37.895,157.149
C03313=1045.509,186.917,404.045,170.932,37.897,157.149
C03314=1045.515,187.166,404.021,170.935,37.900,157.150
C03315=1045.521,187.414,403.997,170.937,37.901,157.150
C03316=1045.527,187.663,403.973,170.940,37.903,157.150
C03317=1045.533,187.912,403.949,170.943,37.905,157.151
C03318=1045.539,188.161,403.925,170.945,37.907,157.151
C03319=1045.545,188.410,403.901,170.947,37.908,157.151
C03320=1045.551,188.659,403.877,170.950,37.910,157.152
C03321=1045.557,188.907,403.852,170.952,37.912,157.152
C03322=1045.563,189.156,403.828,170.955,37.914,157.153
C03323=1045.570,189.440,403.801,170.958,37.916,157.153
C03324=1045.577,189.724,403.773,170.961,37.918,157.154
C03325=1045.583,190.010,403.745,170.964,37.920,157.154
C03326=1045.591,190.294,403.717,170.967,37.923,157.155
C03327=1045.597,190.542,403.693,170.969,37.924,157.155
C03328=1045.603,190.791,403.669,170.972,37.926,157.155
C03329=1045.609,191.040,403.645,170.974,37.928,157.156
C03330=1045.615,191.289,403.621,170.977,37.930,157.156
C03331=1045.620,191.538,403.596,170.980,37.932,157.157
C03332=1045.626,191.787,403.572,170.982,37.934,157.157
C03333=1045.632,192.035,403.547,170.984,37.935,157.158
C03334=1045.639,192.283,403.523,170.988,37.937,157.158
C03335=1045.645,192.533,403.499,170.990,37.939,157.158
C03336=1045.651,192.781,403.475,170.992,37.941,157.159
C03337=1045.657,193.030,403.450,170.996,37.943,157.159
C03338=1045.664,193.279,403.426,170.998,37.945,157.160
C03339=1045.669,193.527,403.401,171.000,37.947,157.160
C03340=1045.675,193.776,403.377,171.003,37.948,157.160
C03341=1045.681,194.024,403.352,171.006,37.950,157.161
C03342=1045.688,194.273,403.328,171.008,37.952,157.161
C03343=1045.694,194.523,403.304,171.011,37.954,157.162
C03344=1045.699,194.771,403.279,171.014,37.956,157.162
C03345=1045.706,195.019,403.255,171.016,37.958,157.163
C03346=1045.712,195.269,403.230,171.019,37.959,157.163
C03347=1045.718,195.517,403.206,171.021,37.962,157.163
C03348=1045.724,195.766,403.181,171.024,37.964,157.164
C03349=1045.731,196.015,403.157,171.027,37.965,157.164
C03350=1045.736,196.263,403.133,171.029,37.967,157.165
C03351=1045.743,196.512,403.108,171.032,37.969,157.165
C03352=1045.749,196.761,403.083,171.035,37.971,157.166
C03353=1045.755,197.010,403.058,171.037,37.973,157.166
C03354=1045.761,197.258,403.034,171.040,37.975,157.166
C03355=1045.767,197.507,403.010,171.043,37.976,157.167
C03356=1045.774,197.755,402.985,171.045,37.979,157.167
C03357=1045.780,198.005,402.960,171.048,37.981,157.168
C03358=1045.786,198.252,402.936,171.051,37.982,157.168
C03359=1045.792,198.502,402.911,171.053,37.984,157.169
C03360=1045.798,198.750,402.886,171.056,37.986,157.169
C03361=1045.805,198.999,402.862,171.059,37.988,157.169
C03362=1045.810,199.247,402.837,171.061,37.990,157.170
C03363=1045.817,199.496,402.813,171.064,37.992,157.170
C03364=1045.823,199.745,402.788,171.067,37.994,157.171
C03365=1045.829,199.994,402.763,171.069,37.996,157.171
C03366=1045.836,200.243,402.738,171.072,37.997,157.172
C03367=1045.841,200.491,402.714,171.075,37.999,157.172
C03368=1045.848,200.740,402.689,171.077,38.002,157.172
C03369=1045.854,200.989,402.665,171.080,38.003,157.173
C03370=1045.860,201.238,402.639,171.083,38.005,157.173
C03371=1045.867,201.486,402.615,171.085,38.007,157.174
C03372=1045.873,201.734,402.590,171.089,38.009,157.174
C03373=1045.879,201.983,402.565,171.091,38.011,157.175
C03374=1045.885,202.232,402.540,171.094,38.013,157.175
C03375=1045.891,202.481,402.515,171.097,38.015,157.176
C03376=1045.897,202.730,402.490,171.099,38.017,157.176
C03377=1045.903,202.978,402.465,171.102,38.019,157.176
C03378=1045.909,203.227,402.440,171.105,38.021,157.177
C03379=1045.915,203.476,402.415,171.107,38.023,157.177
C03380=1045.921,203.724,402.390,171.110,38.026,157.178
C03381=1045.927,203.973,402.364,171.113,38.027,157.178
C03382=1045.933,204.222,402.340,171.115,38.030,157.179
C03383=1045.940,204.470,402.315,171.119,38.031,157.179
C03384=1045.946,204.719,402.290,171.121,38.034,157.180
C03385=1045.952,204.967,402.265,171.124,38.035,157.180
C03386=1045.958,205.216,402.239,171.127,38.038,157.181
C03387=1045.983,206.268,402.132,171.381,38.138,157.206
C03388=1045.991,206.543,402.104,171.382,38.141,157.206
C03389=1045.998,206.817,402.075,171.385,38.144,157.207
C03390=1046.006,207.092,402.046,171.387,38.147,157.208
C03391=1046.013,207.367,402.017,171.389,38.151,157.209
C03392=1046.020,207.616,401.991,171.392,38.153,157.209
C03393=1046.026,207.864,401.965,171.393,38.156,157.210
C03394=1046.033,208.113,401.938,171.396,38.159,157.210
C03395=1046.039,208.361,401.912,171.398,38.162,157.211
C03396=1046.046,208.610,401.885,171.400,38.164,157.212
C03397=1046.052,208.858,401.858,171.402,38.167,157.212
C03398=1046.058,209.107,401.833,171.404,38.170,157.213
C03399=1046.065,209.355,401.807,171.406,38.173,157.214
C03400=1046.071,209.604,401.780,171.408,38.175,157.214
C03401=1046.078,209.852,401.754,171.410,38.178,157.215
C03402=1046.085,210.101,401.728,171.413,38.181,157.215
C03403=1046.091,210.350,401.701,171.414,38.184,157.216
C03404=1046.098,210.598,401.675,171.417,38.187,157.217
C03405=1046.105,210.846,401.648,171.418,38.190,157.217
C03406=1046.111,211.095,401.621,171.421,38.193,157.218
C03407=1046.118,211.343,401.595,171.422,38.196,157.219
C03408=1046.123,211.592,401.568,171.425,38.198,157.219
C03409=1046.131,211.841,401.542,171.427,38.201,157.220
C03410=1046.137,212.089,401.514,171.429,38.204,157.220
C03411=1046.144,212.337,401.488,171.431,38.207,157.221
C03412=1046.150,212.586,401.461,171.433,38.209,157.222
C03413=1046.157,212.834,401.435,171.435,38.212,157.222
C03414=1046.163,213.083,401.408,171.438,38.215,157.223
C03415=1046.170,213.331,401.382,171.440,38.218,157.224
C03416=1046.176,213.580,401.355,171.442,38.220,157.224
C03417=1046.182,213.828,401.329,171.444,38.223,157.225
C03418=1046.189,214.077,401.301,171.446,38.226,157.225
C03419=1046.196,214.325,401.275,171.449,38.229,157.226
C03420=1046.202,214.574,401.248,171.450,38.232,157.227
C03421=1046.208,214.822,401.222,171.453,38.235,157.227
C03422=1046.215,215.071,401.195,171.454,38.238,157.228
C03423=1046.221,215.319,401.168,171.457,38.241,157.229
C03424=1046.228,215.568,401.141,171.459,38.243,157.229
C03425=1046.234,215.817,401.114,171.461,38.246,157.230
C03426=1046.241,216.065,401.088,171.463,38.249,157.230
C03427=1046.248,216.313,401.061,171.466,38.252,157.231
C03428=1046.253,216.561,401.034,171.467,38.254,157.232
C03429=1046.261,216.810,401.007,171.470,38.257,157.232
C03430=1046.267,217.059,400.980,171.472,38.260,157.233
C03431=1046.274,217.307,400.954,171.474,38.262,157.233
C03432=1046.280,217.556,400.927,171.476,38.265,157.234
C03433=1046.286,217.805,400.900,171.479,38.268,157.235
C03434=1046.293,218.052,400.873,171.480,38.271,157.235
C03435=1046.300,218.301,400.846,171.483,38.274,157.236
C03436=1046.306,218.549,400.820,171.485,38.277,157.237
C03437=1046.313,218.798,400.792,171.487,38.280,157.237
C03438=1046.319,219.047,400.765,171.489,38.282,157.238
C03439=1046.326,219.294,400.738,171.492,38.285,157.239
C03440=1046.332,219.543,400.711,171.494,38.288,157.239
C03441=1046.340,219.792,400.685,171.496,38.290,157.240
C03442=1046.346,220.041,400.657,171.499,38.293,157.240
C03443=1046.352,220.289,400.630,171.500,38.296,157.241
C03444=1046.359,220.569,400.600,171.503,38.299,157.242
C03445=1046.367,220.849,400.569,171.505,38.302,157.242
C03446=1046.375,221.129,400.539,171.508,38.305,157.243
C03447=1046.381,221.410,400.508,171.511,38.308,157.244
C03448=1046.388,221.658,400.481,171.513,38.311,157.244
C03449=1046.395,221.907,400.454,171.515,38.314,157.245
C03450=1046.401,222.155,400.427,171.517,38.317,157.246
C03451=1046.407,222.404,400.400,171.520,38.320,157.246
C03452=1046.414,222.652,400.372,171.522,38.323,157.247
C03453=1046.420,222.900,400.345,171.524,38.325,157.248
C03454=1046.427,223.149,400.318,171.526,38.328,157.248
C03455=1046.433,223.397,400.290,171.529,38.331,157.249
C03456=1046.440,223.646,400.264,171.530,38.334,157.250
C03457=1046.446,223.894,400.236,171.533,38.336,157.250
C03458=1046.453,224.142,400.208,171.535,38.339,157.251
C03459=1046.459,224.391,400.181,171.538,38.342,157.251
C03460=1046.466,224.639,400.154,171.539,38.344,157.252
C03461=1046.472,224.888,400.126,171.542,38.347,157.253
C03462=1046.479,225.137,400.099,171.545,38.350,157.253
C03463=1046.485,225.385,400.072,171.547,38.353,157.254
C03464=1046.492,225.633,400.045,171.549,38.355,157.254
C03465=1046.498,225.882,400.018,171.551,38.358,157.255
C03466=1046.505,226.130,399.990,171.554,38.361,157.256
C03467=1046.512,226.379,399.962,171.556,38.364,157.256
C03468=1046.518,226.628,399.935,171.558,38.367,157.257
C03469=1046.524,226.875,399.908,171.560,38.370,157.258
C03470=1046.531,227.124,399.880,171.563,38.372,157.258
C03471=1046.538,227.372,399.853,171.565,38.375,157.259
C03472=1046.544,227.621,399.826,171.567,38.378,157.260
C03473=1046.551,227.869,399.798,171.569,38.380,157.260
C03474=1046.558,228.117,399.771,171.572,38.383,157.261
C03475=1046.564,228.366,399.743,171.574,38.386,157.261
C03476=1046.571,228.614,399.716,171.577,38.388,157.262
C03477=1046.577,228.863,399.689,171.578,38.391,157.263
C03478=1046.584,229.112,399.661,171.581,38.394,157.263
C03479=1046.590,229.359,399.633,171.584,38.396,157.264
C03480=1046.597,229.608,399.606,171.586,38.399,157.264
C03481=1046.603,229.856,399.577,171.589,38.402,157.265
C03482=1046.609,230.105,399.550,171.590,38.405,157.266
C03483=1046.616,230.353,399.522,171.593,38.408,157.266
C03484=1046.623,230.602,399.494,171.595,38.411,157.267
C03485=1046.629,230.849,399.467,171.598,38.413,157.268
C03486=1046.635,231.098,399.439,171.600,38.416,157.268
C03487=1046.642,231.346,399.411,171.602,38.419,157.269
C03488=1046.649,231.595,399.384,171.604,38.422,157.270
C03489=1046.655,231.844,399.355,171.607,38.424,157.270
C03490=1046.661,232.092,399.328,171.609,38.427,157.271
C03491=1046.668,232.340,399.300,171.612,38.430,157.271
C03492=1046.674,232.588,399.273,171.614,38.433,157.272
C03493=1046.681,232.837,399.245,171.616,38.435,157.273
C03494=1046.687,233.085,399.216,171.619,38.438,157.273
C03495=1046.694,233.334,399.189,171.621,38.441,157.274
C03496=1046.700,233.582,399.161,171.624,38.444,157.275
C03497=1046.707,233.831,399.133,171.626,38.446,157.275
C03498=1046.713,234.079,399.105,171.628,38.449,157.276
C03499=1046.720,234.328,399.077,171.630,38.452,157.277
C03500=1046.726,234.600,399.047,171.633,38.455,157.277
C03501=1046.734,234.873,399.016,171.636,38.458,157.278
C03502=1046.741,235.145,398.986,171.638,38.461,157.279
C03503=1046.748,235.418,398.954,171.641,38.464,157.279
C03504=1046.754,235.666,398.926,171.643,38.467,157.280
C03505=1046.761,235.915,398.898,171.646,38.470,157.281
C03506=1046.768,236.163,398.870,171.649,38.472,157.281
C03507=1046.774,236.412,398.843,171.651,38.475,157.282
C03508=1046.781,236.660,398.814,171.654,38.478,157.282
C03509=1046.787,236.908,398.786,171.656,38.481,157.283
C03510=1046.794,237.157,398.758,171.659,38.484,157.284
C03511=1046.800,237.406,398.730,171.660,38.486,157.284
C03512=1046.807,237.653,398.701,171.663,38.489,157.285
C03513=1046.813,237.902,398.674,171.665,38.492,157.286
C03514=1046.820,238.150,398.646,171.668,38.494,157.286
C03515=1046.826,238.399,398.618,171.670,38.497,157.287
C03516=1046.833,238.647,398.589,171.673,38.500,157.288
C03517=1046.840,238.895,398.561,171.675,38.502,157.288
C03518=1046.846,239.144,398.533,171.678,38.505,157.289
C03519=1046.853,239.392,398.505,171.681,38.508,157.289
C03520=1046.859,239.641,398.476,171.683,38.510,157.290
C03521=1046.866,239.888,398.448,171.686,38.513,157.291
C03522=1046.872,240.137,398.420,171.687,38.516,157.291
C03523=1046.878,240.386,398.392,171.690,38.519,157.292
C03524=1046.885,240.633,398.363,171.692,38.521,157.293
C03525=1046.892,240.882,398.336,171.695,38.524,157.293
C03526=1046.898,241.130,398.307,171.697,38.527,157.294
C03527=1046.905,241.378,398.279,171.700,38.529,157.294
C03528=1046.911,241.627,398.250,171.703,38.532,157.295
C03529=1046.918,241.875,398.222,171.705,38.535,157.296
C03530=1046.924,242.123,398.193,171.708,38.538,157.297
C03531=1046.931,242.372,398.165,171.710,38.541,157.297
C03532=1046.937,242.620,398.136,171.713,38.543,157.298
C03533=1046.943,242.868,398.108,171.715,38.546,157.298
C03534=1046.950,243.116,398.080,171.718,38.549,157.299
C03535=1046.956,243.365,398.051,171.720,38.552,157.300
C03536=1046.963,243.613,398.023,171.723,38.554,157.300
C03537=1046.969,243.861,397.994,171.726,38.557,157.301
C03538=1046.975,244.110,397.965,171.728,38.560,157.302
C03539=1046.982,244.358,397.937,171.731,38.563,157.302
C03540=1046.988,244.606,397.908,171.732,38.565,157.303
C03541=1046.996,244.855,397.880,171.735,38.568,157.304
C03542=1047.002,245.103,397.851,171.737,38.571,157.304
C03543=1047.008,245.351,397.822,171.740,38.574,157.305
C03544=1047.015,245.600,397.794,171.743,38.576,157.305
C03545=1047.021,245.848,397.765,171.745,38.579,157.306
C03546=1047.027,246.096,397.736,171.748,38.582,157.307
C03547=1047.033,246.345,397.708,171.750,38.585,157.307
C03548=1047.039,246.593,397.679,171.753,38.588,157.308
C03549=1047.046,246.841,397.650,171.755,38.591,157.309
C03550=1047.053,247.089,397.621,171.758,38.593,157.309
C03551=1047.059,247.337,397.592,171.761,38.596,157.310
C03552=1047.066,247.586,397.563,171.763,38.599,157.311
C03553=1047.072,247.834,397.534,171.766,38.602,157.311
C03554=1047.078,248.083,397.505,171.768,38.605,157.312
C03555=1047.084,248.331,397.476,171.771,38.608,157.313
C03556=1047.091,248.597,397.446,171.774,38.611,157.313
C03557=1047.098,248.864,397.414,171.776,38.614,157.314
C03558=1047.105,249.131,397.383,171.780,38.616,157.315
C03559=1047.112,249.398,397.351,171.782,38.619,157.316
C03560=1047.119,249.646,397.323,171.785,38.622,157.316
C03561=1047.125,249.894,397.294,171.788,38.625,157.317
C03562=1047.131,250.143,397.266,171.790,38.628,157.318
C03563=1047.137,250.391,397.237,171.793,38.631,157.318
C03564=1047.144,250.640,397.207,171.795,38.633,157.319
C03565=1047.150,250.888,397.178,171.798,38.636,157.319
C03566=1047.156,251.136,397.149,171.800,38.639,157.320
C03567=1047.163,251.384,397.120,171.803,38.642,157.321
C03568=1047.169,251.632,397.091,171.806,38.645,157.321
C03569=1047.177,251.881,397.062,171.808,38.648,157.322
C03570=1047.183,252.129,397.033,171.811,38.650,157.323
C03571=1047.189,252.376,397.003,171.813,38.653,157.323
C03572=1047.196,252.625,396.974,171.816,38.656,157.324
C03573=1047.202,252.873,396.945,171.819,38.659,157.325
C03574=1047.209,253.122,396.916,171.822,38.661,157.325
C03575=1047.215,253.370,396.887,171.825,38.664,157.326
C03576=1047.221,253.618,396.858,171.827,38.667,157.327
C03577=1047.228,253.867,396.828,171.830,38.669,157.327
C03578=1047.234,254.115,396.799,171.832,38.672,157.328
C03579=1047.241,254.363,396.771,171.835,38.675,157.329
C03580=1047.248,254.610,396.741,171.838,38.678,157.329
C03581=1047.255,254.859,396.712,171.840,38.680,157.330
C03582=1047.261,255.107,396.683,171.843,38.683,157.331
C03583=1047.267,255.355,396.654,171.845,38.686,157.331
C03584=1047.274,255.604,396.624,171.848,38.689,157.332
C03585=1047.280,255.852,396.595,171.851,38.691,157.333
C03586=1047.287,256.100,396.565,171.854,38.694,157.333
C03587=1047.294,256.349,396.536,171.857,38.697,157.334
C03588=1047.300,256.597,396.507,171.859,38.700,157.335
C03589=1047.306,256.845,396.478,171.862,38.702,157.335
C03590=1047.313,257.093,396.448,171.864,38.705,157.336
C03591=1047.320,257.341,396.419,171.867,38.708,157.337
C03592=1047.326,257.589,396.390,171.871,38.711,157.337
C03593=1047.333,257.837,396.360,171.873,38.714,157.338
C03594=1047.340,258.085,396.331,171.876,38.716,157.338
C03595=1047.347,258.334,396.302,171.878,38.719,157.339
C03596=1047.353,258.582,396.272,171.881,38.722,157.340
C03597=1047.360,258.830,396.243,171.884,38.725,157.341
C03598=1047.366,259.079,396.214,171.887,38.727,157.341
C03599=1047.373,259.326,396.184,171.890,38.730,157.342
C03600=1047.380,259.575,396.154,171.892,38.733,157.342
C03601=1047.386,259.822,396.125,171.895,38.736,157.343
C03602=1047.393,260.071,396.095,171.897,38.738,157.344
C03603=1047.400,260.319,396.066,171.900,38.741,157.344
C03604=1047.406,260.567,396.036,171.904,38.743,157.345
C03605=1047.413,260.816,396.007,171.906,38.746,157.346
C03606=1047.420,261.063,395.977,171.909,38.749,157.346
C03607=1047.426,261.312,395.948,171.911,38.752,157.347
C03608=1047.433,261.560,395.918,171.914,38.754,157.348
C03609=1047.440,261.808,395.889,171.918,38.757,157.348
C03610=1047.446,262.056,395.859,171.920,38.760,157.349
C03611=1047.453,262.305,395.830,171.923,38.762,157.350
C03612=1047.461,262.570,395.798,171.925,38.765,157.350
C03613=1047.467,262.835,395.766,171.929,38.769,157.351
C03614=1047.474,263.101,395.734,171.932,38.772,157.352
C03615=1047.481,263.366,395.702,171.935,38.774,157.353
C03616=1047.487,263.614,395.672,171.938,38.777,157.353
C03617=1047.494,263.863,395.642,171.940,38.780,157.354
C03618=1047.501,264.110,395.613,171.943,38.783,157.355
C03619=1047.507,264.359,395.582,171.946,38.786,157.355
C03620=1047.513,264.607,395.553,171.949,38.789,157.356
C03621=1047.520,264.854,395.523,171.952,38.792,157.357
C03622=1047.526,265.103,395.492,171.955,38.794,157.357
C03623=1047.533,265.350,395.463,171.957,38.797,157.358
C03624=1047.540,265.599,395.433,171.960,38.800,157.359
C03625=1047.546,265.847,395.403,171.963,38.803,157.359
C03626=1047.553,266.095,395.373,171.966,38.805,157.360
C03627=1047.560,266.343,395.343,171.969,38.808,157.361
C03628=1047.566,266.591,395.312,171.971,38.811,157.361
C03629=1047.573,266.840,395.283,171.975,38.814,157.362
C03630=1047.579,267.088,395.253,171.977,38.817,157.363
C03631=1047.585,267.336,395.222,171.980,38.819,157.363
C03632=1047.592,267.584,395.193,171.983,38.822,157.364
C03633=1047.598,267.832,395.162,171.986,38.825,157.365
C03634=1047.605,268.080,395.132,171.989,38.828,157.366
C03635=1047.611,268.328,395.101,171.992,38.831,157.366
C03636=1047.618,268.576,395.072,171.995,38.834,157.367
C03637=1047.625,268.824,395.042,171.998,38.837,157.368
C03638=1047.632,269.072,395.011,172.000,38.839,157.368
C03639=1047.638,269.320,394.981,172.003,38.842,157.369
C03640=1047.645,269.568,394.950,172.007,38.845,157.370
